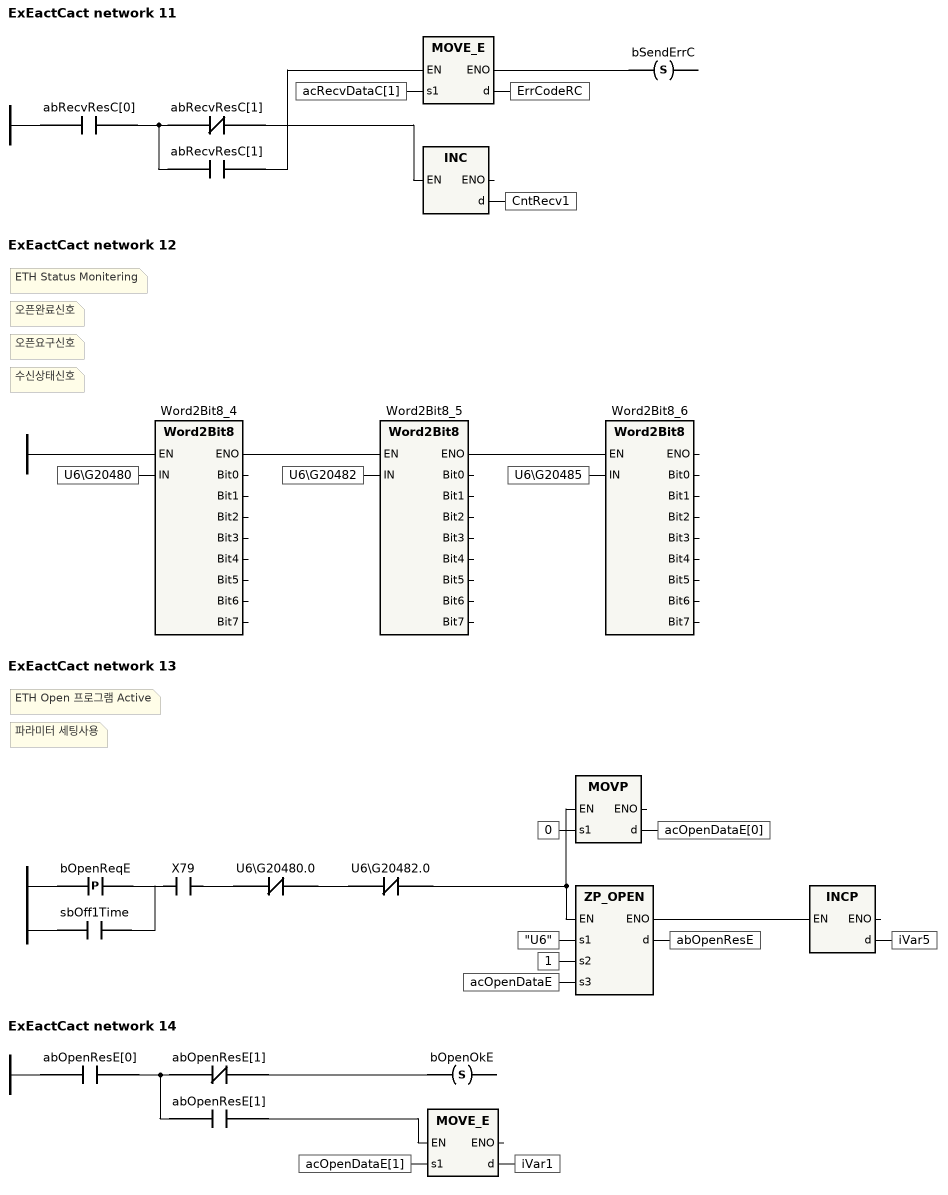
(* [picture p24: structured ladder/FBD of ExEactCact, networks 11 to 14] *)
(* network 11 *)
INC(abRecvResC[0] AND NOT abRecvResC[1], CntRecv1);
_e1 := MOVE_E(abRecvResC[0] AND abRecvResC[1], acRecvDataC[1], ErrCodeRC);
SET(_e1, bSendErrC);
(* network 12 *)
(* ETH Status Monitering *)
(* 오픈완료신호 *)
(* 오픈요구신호 *)
(* 수신상태신호 *)
Word2Bit8_4(EN := TRUE, IN := U6\G20480);
Word2Bit8_5(EN := Word2Bit8_4.ENO, IN := U6\G20482);
Word2Bit8_6(EN := Word2Bit8_5.ENO, IN := U6\G20485);
(* network 13 *)
(* ETH Open 프로그램 Active *)
(* 파라미터 세팅사용 *)
_p1 := (((LDP(TRUE, bOpenReqE) OR sbOff1Time) AND X79) AND NOT U6\G20480.0) AND NOT U6\G20482.0;
MOVP(_p1, 0, acOpenDataE[0]);
_e2 := ZP_OPEN(_p1, "U6", 1, acOpenDataE, abOpenResE);
INCP(_e2, iVar5);
(* network 14 *)
SET(abOpenResE[0] AND NOT abOpenResE[1], bOpenOkE);
MOVE_E(abOpenResE[0] AND abOpenResE[1], acOpenDataE[1], iVar1);
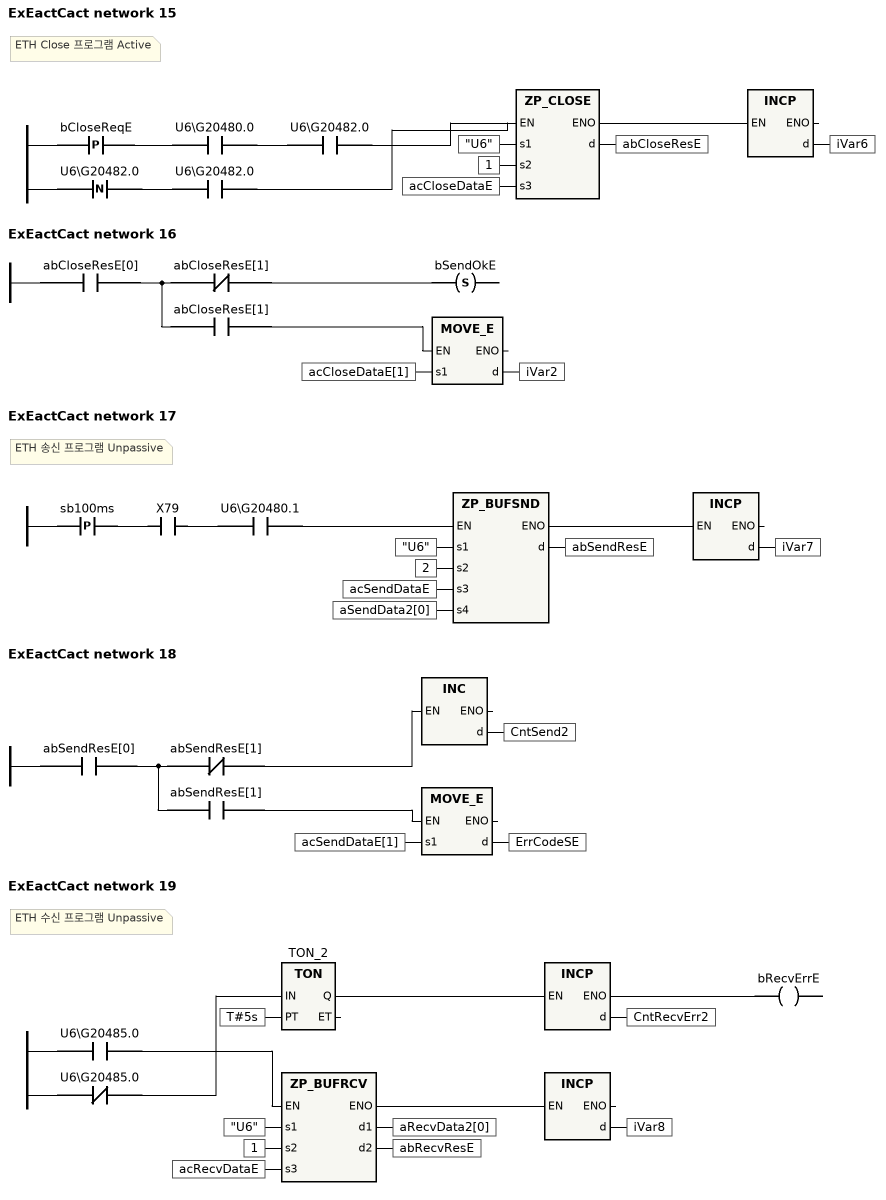
(* network 15 *)
(* ETH Close 프로그램 Active *)
_e1 := ZP_CLOSE((LDP(TRUE, bCloseReqE) AND U6\G20480.0 AND U6\G20482.0) OR (LDF(TRUE, U6\G20482.0) AND U6\G20482.0), "U6", 1, acCloseDataE, abCloseResE);
INCP(_e1, iVar6);
(* network 16 *)
SET(abCloseResE[0] AND NOT abCloseResE[1], bSendOkE);
MOVE_E(abCloseResE[0] AND abCloseResE[1], acCloseDataE[1], iVar2);
(* network 17 *)
(* ETH 송신 프로그램 Unpassive *)
_e1 := ZP_BUFSND(LDP(TRUE, sb100ms) AND X79 AND U6\G20480.1, "U6", 2, acSendDataE, aSendData2[0], abSendResE);
INCP(_e1, iVar7);
(* network 18 *)
INC(abSendResE[0] AND NOT abSendResE[1], CntSend2);
MOVE_E(abSendResE[0] AND abSendResE[1], acSendDataE[1], ErrCodeSE);
(* network 19 *)
(* ETH 수신 프로그램 Unpassive *)
_e1 := ZP_BUFRCV(U6\G20485.0, "U6", 1, acRecvDataE, aRecvData2[0], abRecvResE);
INCP(_e1, iVar8);
TON_2(IN := NOT U6\G20485.0, PT := T#5s);
_e2 := INCP(TON_2.Q, CntRecvErr2);
bRecvErrE := _e2;
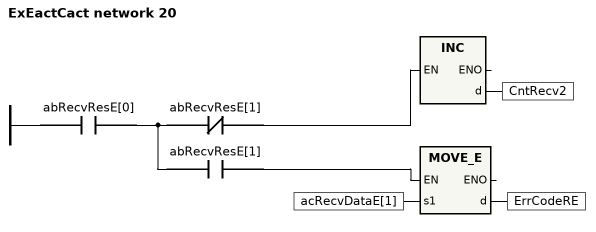
(* network 20 *)
INC(abRecvResE[0] AND NOT abRecvResE[1], CntRecv2);
MOVE_E(abRecvResE[0] AND abRecvResE[1], acRecvDataE[1], ErrCodeRE);
END_PROGRAM

PROGRAM ExEudpCudp
VAR
  bOpenReqC : BOOL;
  bCsetReq : BOOL;
  bOpenReqE : BOOL;
  bOpenOkC : BOOL;
  bOpenOkE : BOOL;
  bOpenErrC : BOOL;
  bOpenErrE : BOOL;
  abOpenResC : ARRAY [0..1] OF BOOL;
  abOpenResE : ARRAY [0..1] OF BOOL;
  acOpenDataC : ARRAY [0..9] OF INT;
  acCsetData : ARRAY [0..4] OF INT;
  acRdCtrl : ARRAY [0..9] OF INT;
  bSendReqC : BOOL;
  bSendReqE : BOOL;
  bSendOkC : BOOL;
  bSendOkE : BOOL;
  bSendErrC : BOOL;
  bSendErrE : BOOL;
  abSendResC : ARRAY [0..1] OF BOOL;
  abSendResE : ARRAY [0..1] OF BOOL;
  abSendResF : ARRAY [0..1] OF BOOL;
  acSendDataC : ARRAY [0..1] OF INT;
  acSendDataE : ARRAY [0..1] OF INT;
  acSendDataF : ARRAY [0..1] OF INT;
  bRecvOkC : BOOL;
  bRecvOkE : BOOL;
  bRecvOkF : BOOL;
  bRecvErrC : BOOL;
  bRecvErrE : BOOL;
  bRecvErrF : BOOL;
  abRecvResC : ARRAY [0..1] OF BOOL;
  abRecvRes3 : ARRAY [0..1] OF BOOL;
  abRecvRes13 : ARRAY [0..1] OF BOOL;
  acRecvDataC : ARRAY [0..1] OF INT;
  acRecvData3 : ARRAY [0..1] OF INT;
  acRecvData13 : ARRAY [0..1] OF INT;
  bCloseReqC : BOOL;
  bCloseOkC : BOOL;
  bCloseOkE : BOOL;
  bCloseErrC : BOOL;
  bCloseErrE : BOOL;
  abCloseResC : ARRAY [0..1] OF BOOL;
  abCloseResE : ARRAY [0..1] OF BOOL;
  acCloseDataC : ARRAY [0..1] OF INT;
  CntSend1 : INT;
  CntSend2 : INT;
  CntSend3 : INT;
  CntRecv1 : INT;
  CntRecvErr1 : INT;
  CntRecv2 : INT;
  CntRecv3 : INT;
  CntRecvErr2 : INT;
  CntRecvErr3 : INT;
  ErrCodeSC : INT;
  ErrCodeSE : INT;
  ErrCodeSF : INT;
  ErrCodeRC : INT;
  ErrCodeR3 : INT;
  ErrCodeR13 : INT;
  Mov4INT_1 : Mov4INT;
  Mov8INT_1 : Mov8INT;
  Mov4INT_2 : Mov4INT;
  Mov4INT_3 : Mov4INT;
  Mov4INT_4 : Mov4INT;
  Word2Bit8_1 : Word2Bit8;
  Word2Bit8_2 : Word2Bit8;
  Word2Bit8_3 : Word2Bit8;
  Word2Bit8_4 : Word2Bit8;
  Word2Bit8_5 : Word2Bit8;
  Word2Bit8_6 : Word2Bit8;
  TON_1 : TON;
  TON_2 : TON;
  TON_3 : TON;
  bCloseReqE : BOOL;
  acOpenDataE : ARRAY [0..9] OF INT;
  acCloseDataE : ARRAY [0..1] OF INT;
  ErrCodeOC : INT;
  ErrCodeOE : INT;
  ErrCodeCC : INT;
  ErrCodeCE : INT;
  bDelay : BOOL;
  bLedOff : BOOL;
  bChgReq : BOOL;
  bChgConn : BOOL;
  ChgPort : INT;
  CntRecv13 : INT;
  TON_13 : TON;
END_VAR
(* structured ladder/FBD written out as ST: instructions are called as NAME(EN, inputs, outputs); _pN, _eN, _tN stand for wires *)
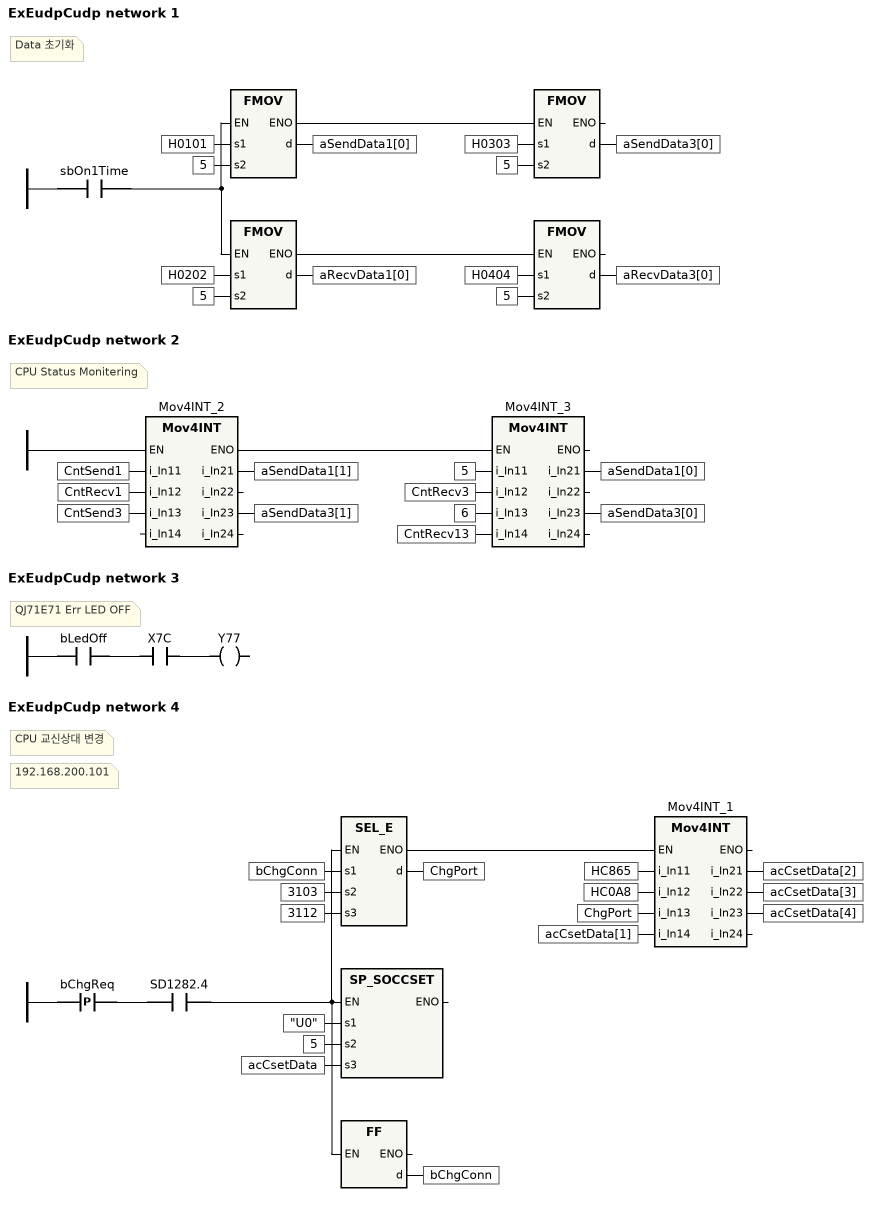
(* network 1 *)
(* Data 초기화 *)
_e1 := FMOV(sbOn1Time, H0101, 5, aSendData1[0]);
FMOV(_e1, H0303, 5, aSendData3[0]);
_e2 := FMOV(sbOn1Time, H0202, 5, aRecvData1[0]);
FMOV(_e2, H0404, 5, aRecvData3[0]);
(* network 2 *)
(* CPU Status Monitering *)
Mov4INT_2(EN := TRUE, i_In11 := CntSend1, i_In12 := CntRecv1, i_In13 := CntSend3, i_In21 => aSendData1[1], i_In23 => aSendData3[1]);
Mov4INT_3(EN := Mov4INT_2.ENO, i_In11 := 5, i_In12 := CntRecv3, i_In13 := 6, i_In14 := CntRecv13, i_In21 => aSendData1[0], i_In23 => aSendData3[0]);
(* network 3 *)
(* QJ71E71 Err LED OFF *)
Y77 := bLedOff AND X7C;
(* network 4 *)
(* CPU 교신상대 변경 *)
(* 192.168.200.101 *)
_p1 := LDP(TRUE, bChgReq) AND SD1282.4;
_e2 := SEL_E(_p1, bChgConn, 3103, 3112, ChgPort);
Mov4INT_1(EN := _e2, i_In11 := HC865, i_In12 := HC0A8, i_In13 := ChgPort, i_In14 := acCsetData[1], i_In21 => acCsetData[2], i_In22 => acCsetData[3], i_In23 => acCsetData[4]);
SP_SOCCSET(_p1, "U0", 5, acCsetData);
FF(_p1, bChgConn);
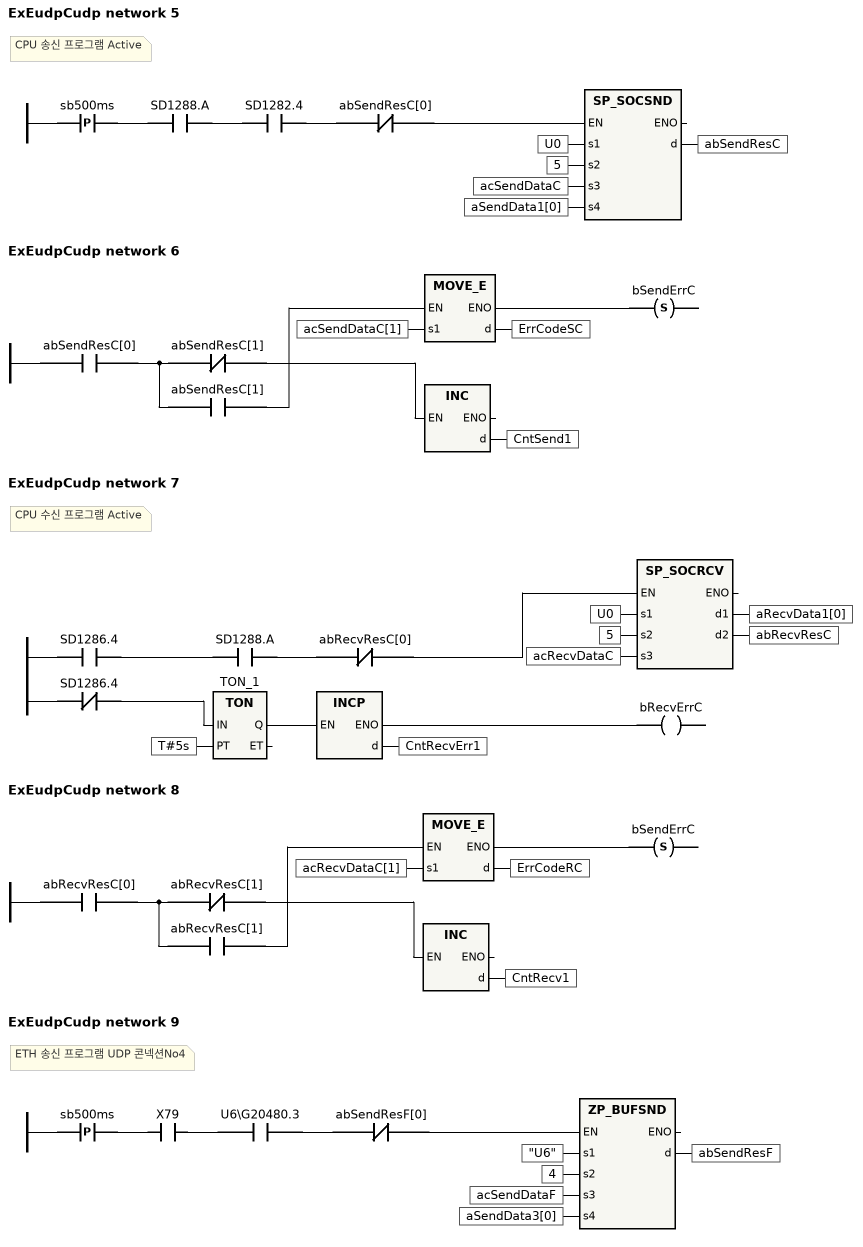
(* network 5 *)
(* CPU 송신 프로그램 Active *)
SP_SOCSND(LDP(TRUE, sb500ms) AND SD1288.A AND SD1282.4 AND NOT abSendResC[0], U0, 5, acSendDataC, aSendData1[0], abSendResC);
(* network 6 *)
INC(abSendResC[0] AND NOT abSendResC[1], CntSend1);
_e1 := MOVE_E(abSendResC[0] AND abSendResC[1], acSendDataC[1], ErrCodeSC);
SET(_e1, bSendErrC);
(* network 7 *)
(* CPU 수신 프로그램 Active *)
SP_SOCRCV(SD1286.4 AND SD1288.A AND NOT abRecvResC[0], U0, 5, acRecvDataC, aRecvData1[0], abRecvResC);
TON_1(IN := NOT SD1286.4, PT := T#5s);
_e1 := INCP(TON_1.Q, CntRecvErr1);
bRecvErrC := _e1;
(* network 8 *)
INC(abRecvResC[0] AND NOT abRecvResC[1], CntRecv1);
_e1 := MOVE_E(abRecvResC[0] AND abRecvResC[1], acRecvDataC[1], ErrCodeRC);
SET(_e1, bSendErrC);
(* network 9 *)
(* ETH 송신 프로그램 UDP 콘넥션No4 *)
ZP_BUFSND(LDP(TRUE, sb500ms) AND X79 AND U6\G20480.3 AND NOT abSendResF[0], "U6", 4, acSendDataF, aSendData3[0], abSendResF);
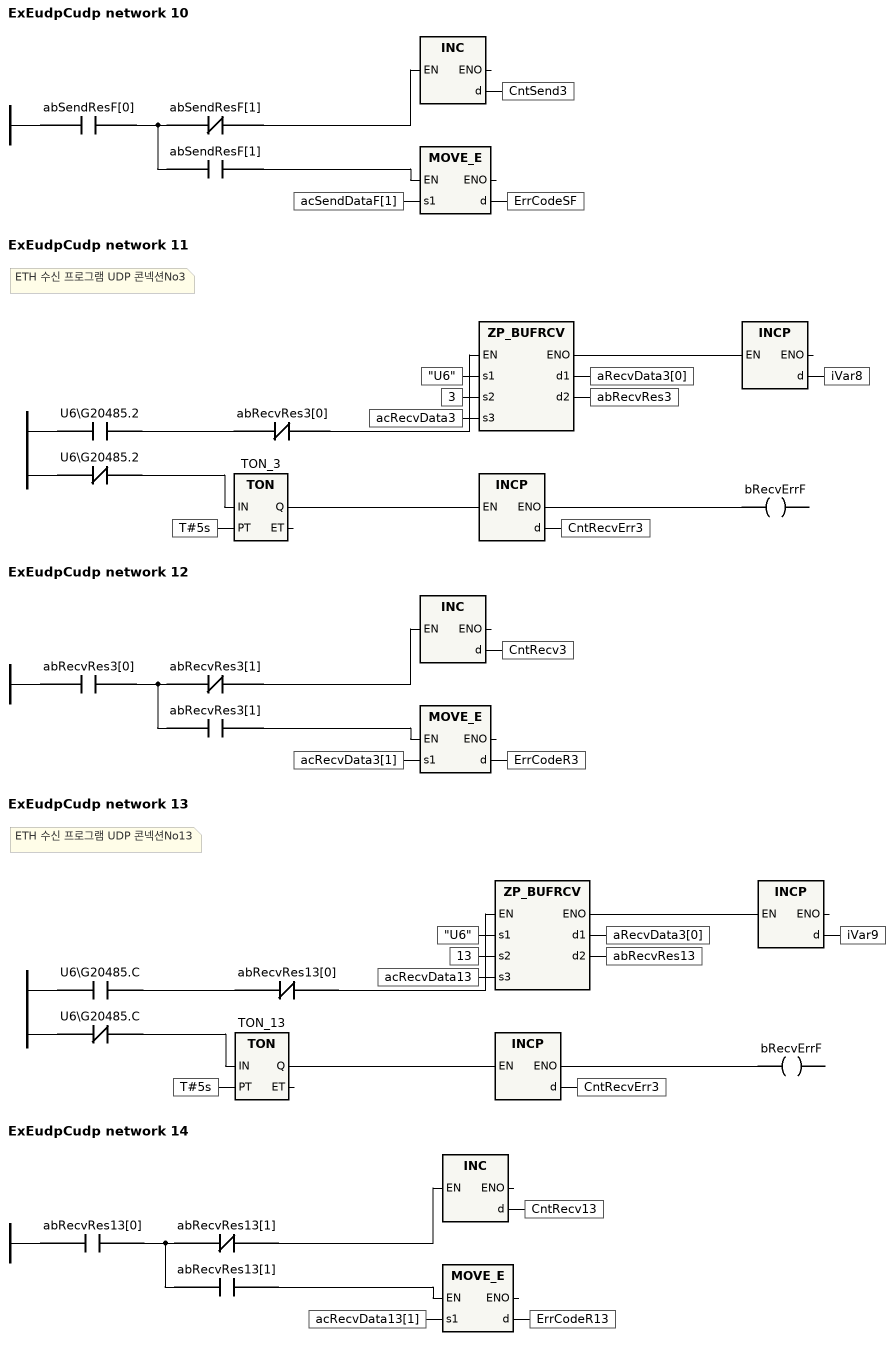
(* network 10 *)
INC(abSendResF[0] AND NOT abSendResF[1], CntSend3);
MOVE_E(abSendResF[0] AND abSendResF[1], acSendDataF[1], ErrCodeSF);
(* network 11 *)
(* ETH 수신 프로그램 UDP 콘넥션No3 *)
_e1 := ZP_BUFRCV(U6\G20485.2 AND NOT abRecvRes3[0], "U6", 3, acRecvData3, aRecvData3[0], abRecvRes3);
INCP(_e1, iVar8);
TON_3(IN := NOT U6\G20485.2, PT := T#5s);
_e2 := INCP(TON_3.Q, CntRecvErr3);
bRecvErrF := _e2;
(* network 12 *)
INC(abRecvRes3[0] AND NOT abRecvRes3[1], CntRecv3);
MOVE_E(abRecvRes3[0] AND abRecvRes3[1], acRecvData3[1], ErrCodeR3);
(* network 13 *)
(* ETH 수신 프로그램 UDP 콘넥션No13 *)
_e1 := ZP_BUFRCV(U6\G20485.C AND NOT abRecvRes13[0], "U6", 13, acRecvData13, aRecvData3[0], abRecvRes13);
INCP(_e1, iVar9);
TON_13(IN := NOT U6\G20485.C, PT := T#5s);
_e2 := INCP(TON_13.Q, CntRecvErr3);
bRecvErrF := _e2;
(* network 14 *)
INC(abRecvRes13[0] AND NOT abRecvRes13[1], CntRecv13);
MOVE_E(abRecvRes13[0] AND abRecvRes13[1], acRecvData13[1], ErrCodeR13);
END_PROGRAM

FUNCTION_BLOCK Word2Bit16
VAR_INPUT
  bEN : BOOL;
END_VAR
VAR_OUTPUT
  Bit0 : BOOL;
  Bit1 : BOOL;
  Bit2 : BOOL;
  Bit3 : BOOL;
  Bit4 : BOOL;
  Bit5 : BOOL;
  Bit6 : BOOL;
  Bit7 : BOOL;
  Bit8 : BOOL;
  Bit9 : BOOL;
  Bit10 : BOOL;
  Bit11 : BOOL;
  Bit12 : BOOL;
  Bit13 : BOOL;
  Bit14 : BOOL;
  Bit15 : BOOL;
END_VAR
VAR_INPUT
  InWord : WORD;
END_VAR
VAR_OUTPUT
  bENO : BOOL;
END_VAR
VAR
  InVal : WORD;
END_VAR
 
bENO := bEN;
InVal :=InWord;
Bit0 := (InVal AND 16#0001) = H0001;
Bit1 := (InVal AND 16#0002) = H0002;
Bit2 := (InVal AND 16#0004) = H0004;
Bit3 := (InVal AND 16#0008) = H0008;
Bit4 := (InVal AND 16#0010) = H0010;
Bit5 := (InVal AND 16#0020) = H0020;
Bit6 := (InVal AND 16#0040) = H0040;
Bit7 := (InVal AND 16#0080) = H0080;
Bit8 := (InVal AND 16#0100) = H0100;
Bit9 := (InVal AND 16#0200) = H0200;
Bit10 := (InVal AND 16#0400) = H0400;
Bit11 := (InVal AND 16#0800) = H0800;
Bit12 := (InVal AND 16#1000) = H1000;
Bit13 := (InVal AND 16#2000) = H2000;
Bit14 := (InVal AND 16#4000) = H4000;
Bit15 := (InVal AND 16#8000) = H8000;

(*
Bit0 := WORD_TO_BOOL(IN AND 16#0001);
Bit1 := WORD_TO_BOOL(SHR(IN AND 16#0002 , 1));
Bit2 := WORD_TO_BOOL(SHR(IN AND 16#0004 , 2));
Bit3 := WORD_TO_BOOL(SHR(IN AND 16#0008 , 3));
Bit4 := WORD_TO_BOOL(SHR(IN AND 16#0010 , 4));
Bit5 := WORD_TO_BOOL(SHR(IN AND 16#0020 , 5));
Bit6 := WORD_TO_BOOL(SHR(IN AND 16#0040 , 6));
Bit7 := WORD_TO_BOOL(SHR(IN AND 16#0080 , 7));
 
Bit8 := WORD_TO_BOOL(SHR(IN AND 16#0100 , 8));
Bit9 := WORD_TO_BOOL(SHR(IN AND 16#0200 , 9));
Bit10 := WORD_TO_BOOL(SHR(IN AND 16#0400 , 10));
Bit11 := WORD_TO_BOOL(SHR(IN AND 16#0800 , 11));
Bit12 := WORD_TO_BOOL(SHR(IN AND 16#1000 , 12));
Bit13 := WORD_TO_BOOL(SHR(IN AND 16#2000 , 13));
Bit14 := WORD_TO_BOOL(SHR(IN AND 16#4000 , 14));
Bit15 := WORD_TO_BOOL(SHR(IN AND 16#8000 , 15));
*)
END_FUNCTION_BLOCK

PROGRAM ExEactCpas
VAR
  bOpenReqC : BOOL;
  bCsetReq : BOOL;
  bOpenReqE : BOOL;
  bOpenOkC : BOOL;
  bOpenOkE : BOOL;
  bOpenErrC : BOOL;
  bOpenErrE : BOOL;
  abOpenResC : ARRAY [0..1] OF BOOL;
  abOpenResE : ARRAY [0..1] OF BOOL;
  acOpenDataC : ARRAY [0..9] OF INT;
  acCsetData : ARRAY [0..4] OF INT;
  acRdCtrl : ARRAY [0..9] OF INT;
  bSendReqC : BOOL;
  bSendReqE : BOOL;
  bSendOkC : BOOL;
  bSendOkE : BOOL;
  bSendErrC : BOOL;
  bSendErrE : BOOL;
  abSendResC : ARRAY [0..1] OF BOOL;
  abSendResE : ARRAY [0..1] OF BOOL;
  abSendResF : ARRAY [0..1] OF BOOL;
  acSendDataC : ARRAY [0..1] OF INT;
  acSendDataE : ARRAY [0..1] OF INT;
  acSendDataF : ARRAY [0..1] OF INT;
  bRecvOkC : BOOL;
  bRecvOkE : BOOL;
  bRecvOkF : BOOL;
  bRecvErrC : BOOL;
  bRecvErrE : BOOL;
  bRecvErrF : BOOL;
  abRecvResC : ARRAY [0..1] OF BOOL;
  abRecvResE : ARRAY [0..1] OF BOOL;
  abRecvResF : ARRAY [0..1] OF BOOL;
  acRecvDataC : ARRAY [0..1] OF INT;
  acRecvDataE : ARRAY [0..1] OF INT;
  acRecvDataF : ARRAY [0..1] OF INT;
  bCloseReqC : BOOL;
  bCloseOkC : BOOL;
  bCloseOkE : BOOL;
  bCloseErrC : BOOL;
  bCloseErrE : BOOL;
  abCloseResC : ARRAY [0..1] OF BOOL;
  abCloseResE : ARRAY [0..1] OF BOOL;
  acCloseDataC : ARRAY [0..1] OF INT;
  CntSend1 : INT;
  CntSend2 : INT;
  CntSend3 : INT;
  CntRecv1 : INT;
  CntRecvErr1 : INT;
  CntRecv2 : INT;
  CntRecv3 : INT;
  CntRecvErr2 : INT;
  CntRecvErr3 : INT;
  ErrCodeCC : INT;
  ErrCodeSE : INT;
  ErrCodeSF : INT;
  ErrCodeRC : INT;
  ErrCodeRE : INT;
  ErrCodeRF : INT;
  Mov4INT_1 : Mov4INT;
  Mov8INT_1 : Mov8INT;
  Mov4INT_2 : Mov4INT;
  Mov4INT_3 : Mov4INT;
  Mov4INT_4 : Mov4INT;
  Word2Bit8_1 : Word2Bit8;
  Word2Bit8_2 : Word2Bit8;
  Word2Bit8_3 : Word2Bit8;
  Word2Bit8_4 : Word2Bit8;
  Word2Bit8_5 : Word2Bit8;
  Word2Bit8_6 : Word2Bit8;
  TON_1 : TON;
  TON_2 : TON;
  TON_3 : TON;
  Status1 : WORD;
  Status2 : WORD;
  Status3 : WORD;
  Word2Bit16_1 : Word2Bit16;
  Word2Bit16_2 : Word2Bit16;
  Word2Bit16_3 : Word2Bit16;
  acOpenDataE : ARRAY [0..9] OF INT;
  acCloseDataE : ARRAY [0..1] OF INT;
  ErrCodeOE : INT;
  ErrCodeSC : INT;
  ErrCodeCE : INT;
  ErrCodeOC : INT;
  bCloseReqE : BOOL;
  Mov4INT_5 : Mov4INT;
  Mov4INT_6 : Mov4INT;
  Mov4INT_7 : Mov4INT;
  Mov4INT_8 : Mov4INT;
END_VAR
(* structured ladder/FBD written out as ST: instructions are called as NAME(EN, inputs, outputs); _pN, _eN, _tN stand for wires *)
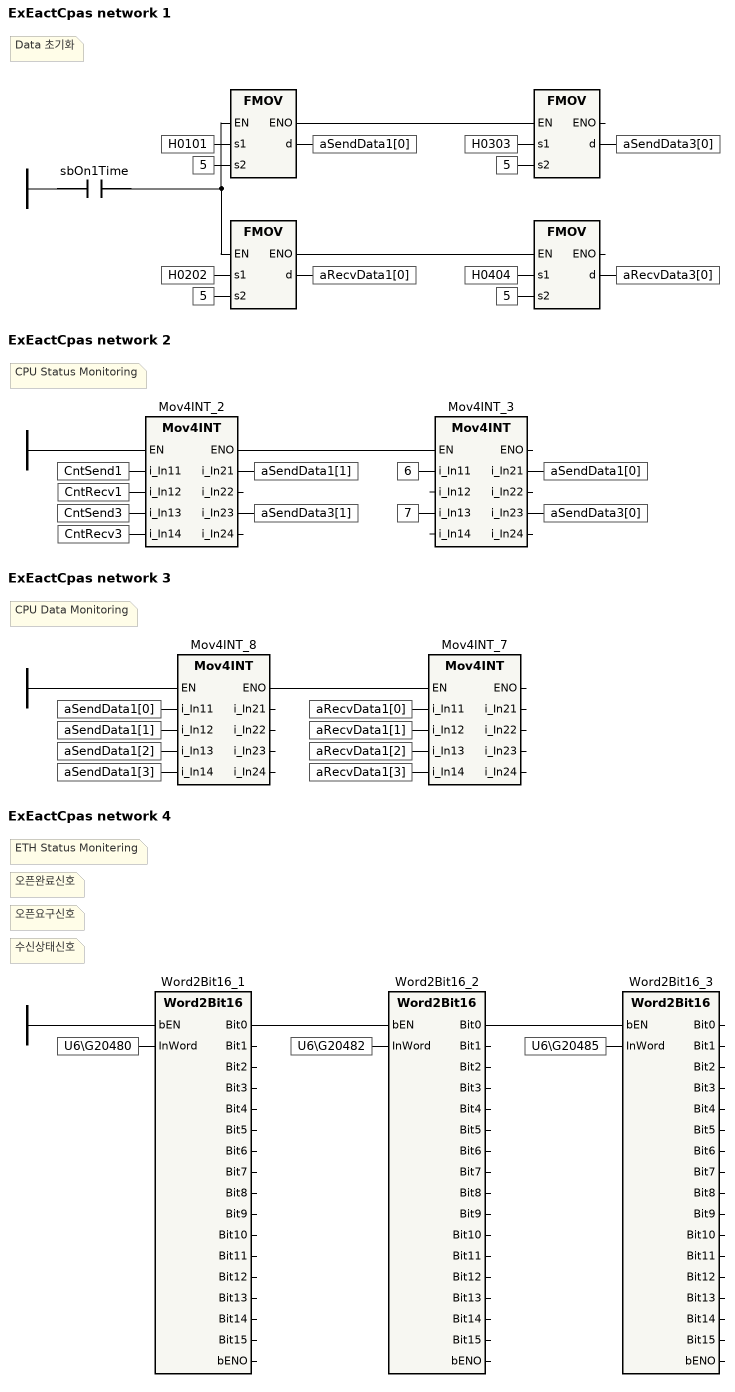
(* network 1 *)
(* Data 초기화 *)
_e1 := FMOV(sbOn1Time, H0101, 5, aSendData1[0]);
FMOV(_e1, H0303, 5, aSendData3[0]);
_e2 := FMOV(sbOn1Time, H0202, 5, aRecvData1[0]);
FMOV(_e2, H0404, 5, aRecvData3[0]);
(* network 2 *)
(* CPU Status Monitoring *)
Mov4INT_2(EN := TRUE, i_In11 := CntSend1, i_In12 := CntRecv1, i_In13 := CntSend3, i_In14 := CntRecv3, i_In21 => aSendData1[1], i_In23 => aSendData3[1]);
Mov4INT_3(EN := Mov4INT_2.ENO, i_In11 := 6, i_In13 := 7, i_In21 => aSendData1[0], i_In23 => aSendData3[0]);
(* network 3 *)
(* CPU Data Monitoring *)
Mov4INT_8(EN := TRUE, i_In11 := aSendData1[0], i_In12 := aSendData1[1], i_In13 := aSendData1[2], i_In14 := aSendData1[3]);
Mov4INT_7(EN := Mov4INT_8.ENO, i_In11 := aRecvData1[0], i_In12 := aRecvData1[1], i_In13 := aRecvData1[2], i_In14 := aRecvData1[3]);
(* network 4 *)
(* ETH Status Monitering *)
(* 오픈완료신호 *)
(* 오픈요구신호 *)
(* 수신상태신호 *)
Word2Bit16_1(bEN := TRUE, InWord := U6\G20480);
Word2Bit16_2(bEN := Word2Bit16_1.Bit0, InWord := U6\G20482);
Word2Bit16_3(bEN := Word2Bit16_2.Bit0, InWord := U6\G20485);
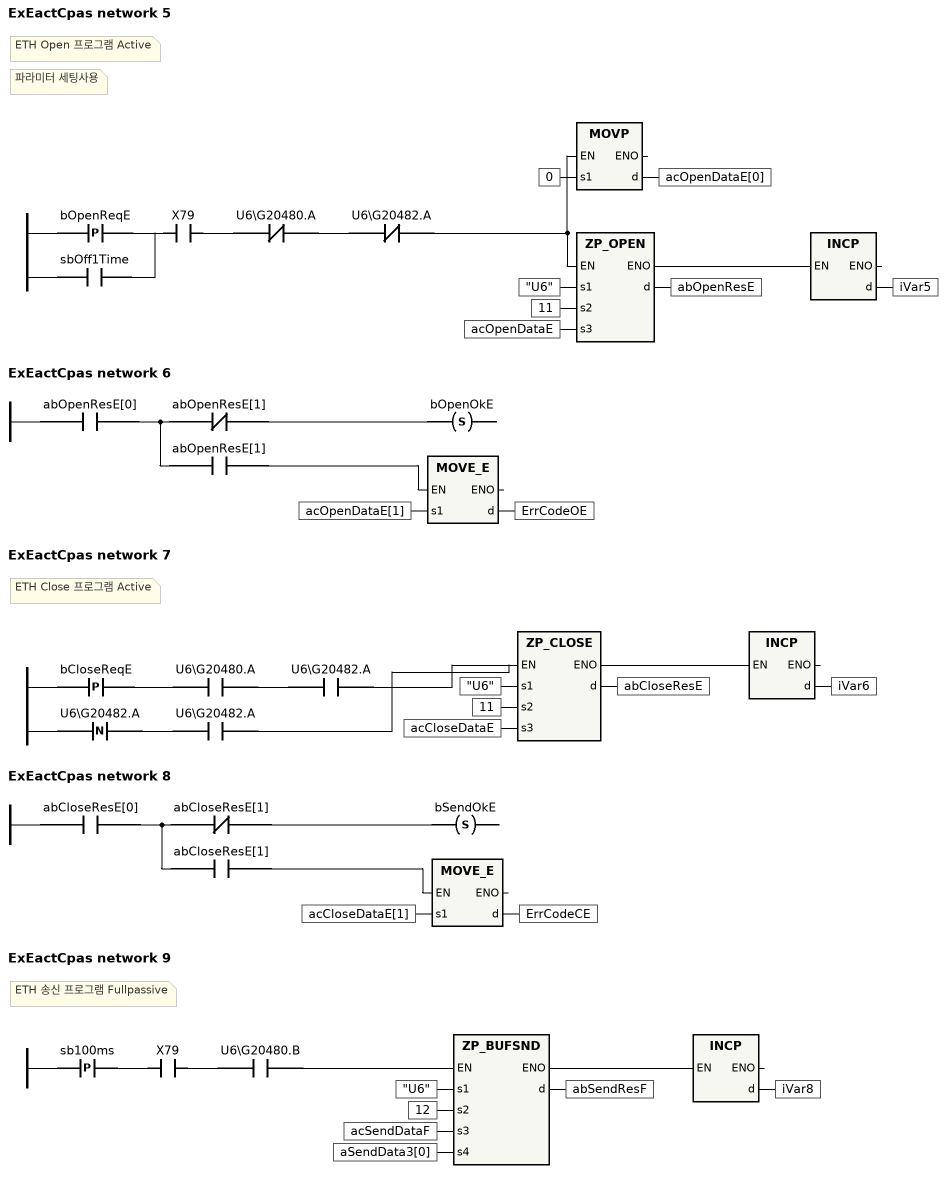
(* network 5 *)
(* ETH Open 프로그램 Active *)
(* 파라미터 세팅사용 *)
_p1 := (((LDP(TRUE, bOpenReqE) OR sbOff1Time) AND X79) AND NOT U6\G20480.A) AND NOT U6\G20482.A;
MOVP(_p1, 0, acOpenDataE[0]);
_e2 := ZP_OPEN(_p1, "U6", 11, acOpenDataE, abOpenResE);
INCP(_e2, iVar5);
(* network 6 *)
SET(abOpenResE[0] AND NOT abOpenResE[1], bOpenOkE);
MOVE_E(abOpenResE[0] AND abOpenResE[1], acOpenDataE[1], ErrCodeOE);
(* network 7 *)
(* ETH Close 프로그램 Active *)
_e1 := ZP_CLOSE((LDP(TRUE, bCloseReqE) AND U6\G20480.A AND U6\G20482.A) OR (LDF(TRUE, U6\G20482.A) AND U6\G20482.A), "U6", 11, acCloseDataE, abCloseResE);
INCP(_e1, iVar6);
(* network 8 *)
SET(abCloseResE[0] AND NOT abCloseResE[1], bSendOkE);
MOVE_E(abCloseResE[0] AND abCloseResE[1], acCloseDataE[1], ErrCodeCE);
(* network 9 *)
(* ETH 송신 프로그램 Fullpassive *)
_e1 := ZP_BUFSND(LDP(TRUE, sb100ms) AND X79 AND U6\G20480.B, "U6", 12, acSendDataF, aSendData3[0], abSendResF);
INCP(_e1, iVar8);
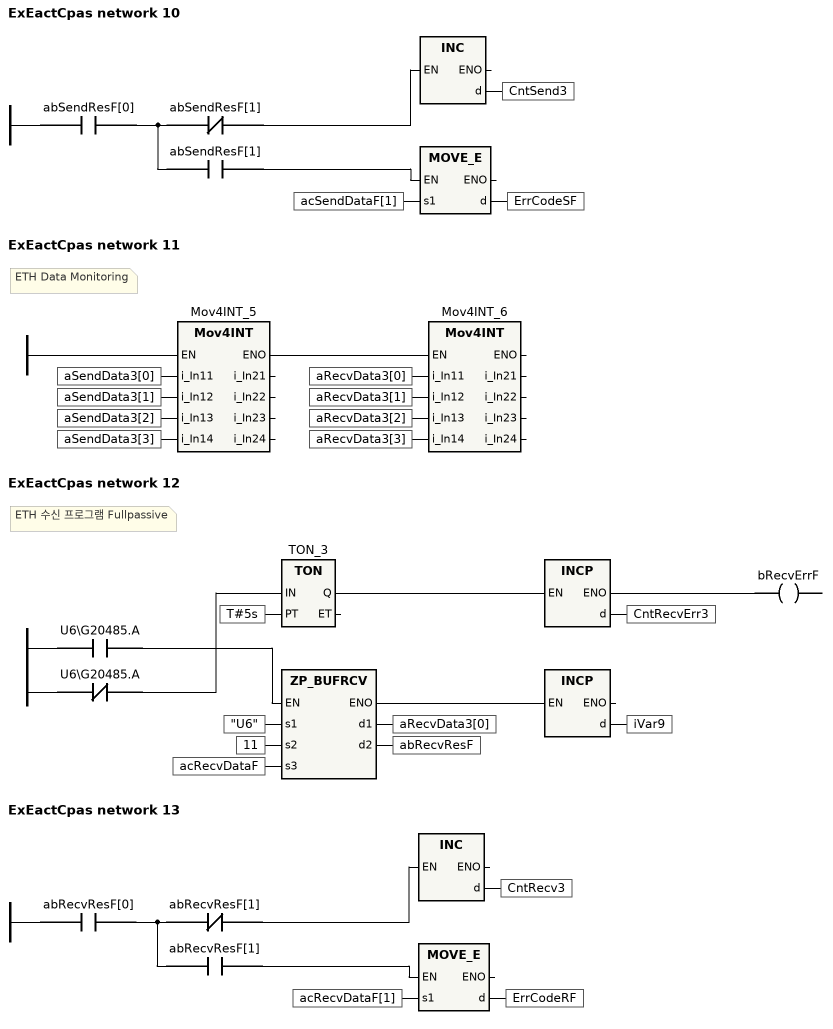
(* network 10 *)
INC(abSendResF[0] AND NOT abSendResF[1], CntSend3);
MOVE_E(abSendResF[0] AND abSendResF[1], acSendDataF[1], ErrCodeSF);
(* network 11 *)
(* ETH Data Monitoring *)
Mov4INT_5(EN := TRUE, i_In11 := aSendData3[0], i_In12 := aSendData3[1], i_In13 := aSendData3[2], i_In14 := aSendData3[3]);
Mov4INT_6(EN := Mov4INT_5.ENO, i_In11 := aRecvData3[0], i_In12 := aRecvData3[1], i_In13 := aRecvData3[2], i_In14 := aRecvData3[3]);
(* network 12 *)
(* ETH 수신 프로그램 Fullpassive *)
_e1 := ZP_BUFRCV(U6\G20485.A, "U6", 11, acRecvDataF, aRecvData3[0], abRecvResF);
INCP(_e1, iVar9);
TON_3(IN := NOT U6\G20485.A, PT := T#5s);
_e2 := INCP(TON_3.Q, CntRecvErr3);
bRecvErrF := _e2;
(* network 13 *)
INC(abRecvResF[0] AND NOT abRecvResF[1], CntRecv3);
MOVE_E(abRecvResF[0] AND abRecvResF[1], acRecvDataF[1], ErrCodeRF);
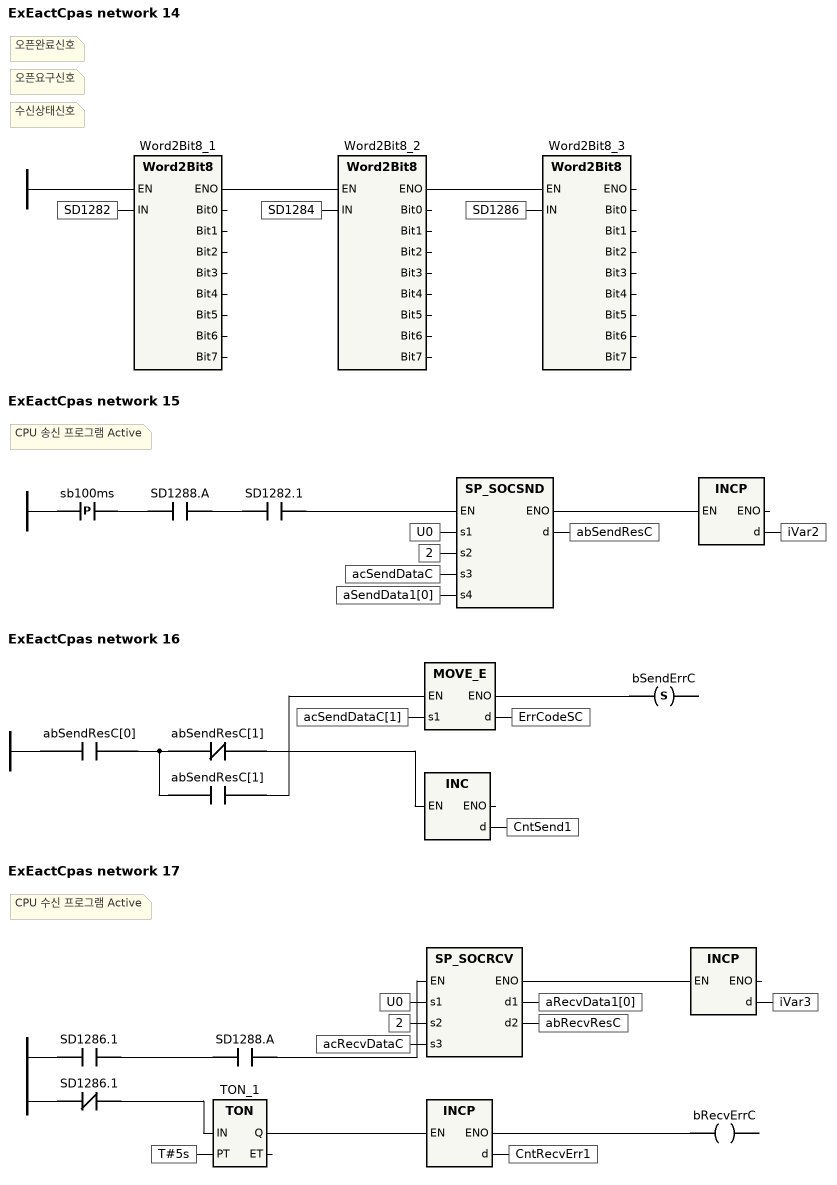
(* network 14 *)
(* 오픈완료신호 *)
(* 오픈요구신호 *)
(* 수신상태신호 *)
Word2Bit8_1(EN := TRUE, IN := SD1282);
Word2Bit8_2(EN := Word2Bit8_1.ENO, IN := SD1284);
Word2Bit8_3(EN := Word2Bit8_2.ENO, IN := SD1286);
(* network 15 *)
(* CPU 송신 프로그램 Active *)
_e1 := SP_SOCSND(LDP(TRUE, sb100ms) AND SD1288.A AND SD1282.1, U0, 2, acSendDataC, aSendData1[0], abSendResC);
INCP(_e1, iVar2);
(* network 16 *)
INC(abSendResC[0] AND NOT abSendResC[1], CntSend1);
_e1 := MOVE_E(abSendResC[0] AND abSendResC[1], acSendDataC[1], ErrCodeSC);
SET(_e1, bSendErrC);
(* network 17 *)
(* CPU 수신 프로그램 Active *)
_e1 := SP_SOCRCV(SD1286.1 AND SD1288.A, U0, 2, acRecvDataC, aRecvData1[0], abRecvResC);
INCP(_e1, iVar3);
TON_1(IN := NOT SD1286.1, PT := T#5s);
_e2 := INCP(TON_1.Q, CntRecvErr1);
bRecvErrC := _e2;
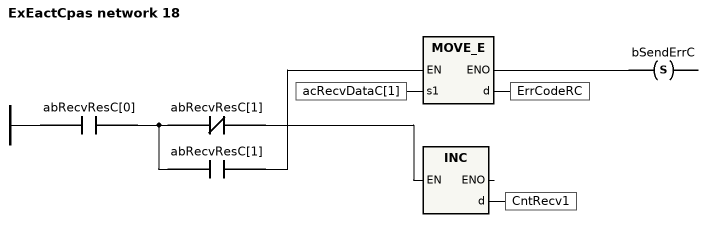
(* network 18 *)
INC(abRecvResC[0] AND NOT abRecvResC[1], CntRecv1);
_e1 := MOVE_E(abRecvResC[0] AND abRecvResC[1], acRecvDataC[1], ErrCodeRC);
SET(_e1, bSendErrC);
END_PROGRAM

PROGRAM ExZP_OPEN
VAR
  bOpenExeE : BOOL;
  bOpenOkE : BOOL;
  bOpenErrE : BOOL;
  bComp11 : BOOL;
  bReq11 : BOOL;
  acOpenDataE : ARRAY [0..9] OF INT;
  bCloseTime : BOOL;
  bCloseReqE : BOOL;
  bCloseExeE : BOOL;
  bCloseReqA : BOOL;
  bCloseIng : BOOL;
  acCloseDataE : ARRAY [0..1] OF INT;
  abOpenResE : ARRAY [0..1] OF BOOL;
  abCloseResE : ARRAY [0..1] OF BOOL;
  bCloseOkE : BOOL;
  bCloseErrE : BOOL;
  bOpenReqM : BOOL;
  bCloseReqM : BOOL;
  Word2Bit16_1 : Word2Bit16;
  Word2Bit16_2 : Word2Bit16;
  Word2Bit16_3 : Word2Bit16;
  abSendResE : ARRAY [0..1] OF BOOL;
  acSendDataE : ARRAY [0..1] OF INT;
  Mov4INT_1 : Mov4INT;
  bReqFlag : BOOL;
  bFlagExe : BOOL;
  bReqOpen : BOOL;
END_VAR
(* structured ladder/FBD written out as ST: instructions are called as NAME(EN, inputs, outputs); _pN, _eN, _tN stand for wires *)
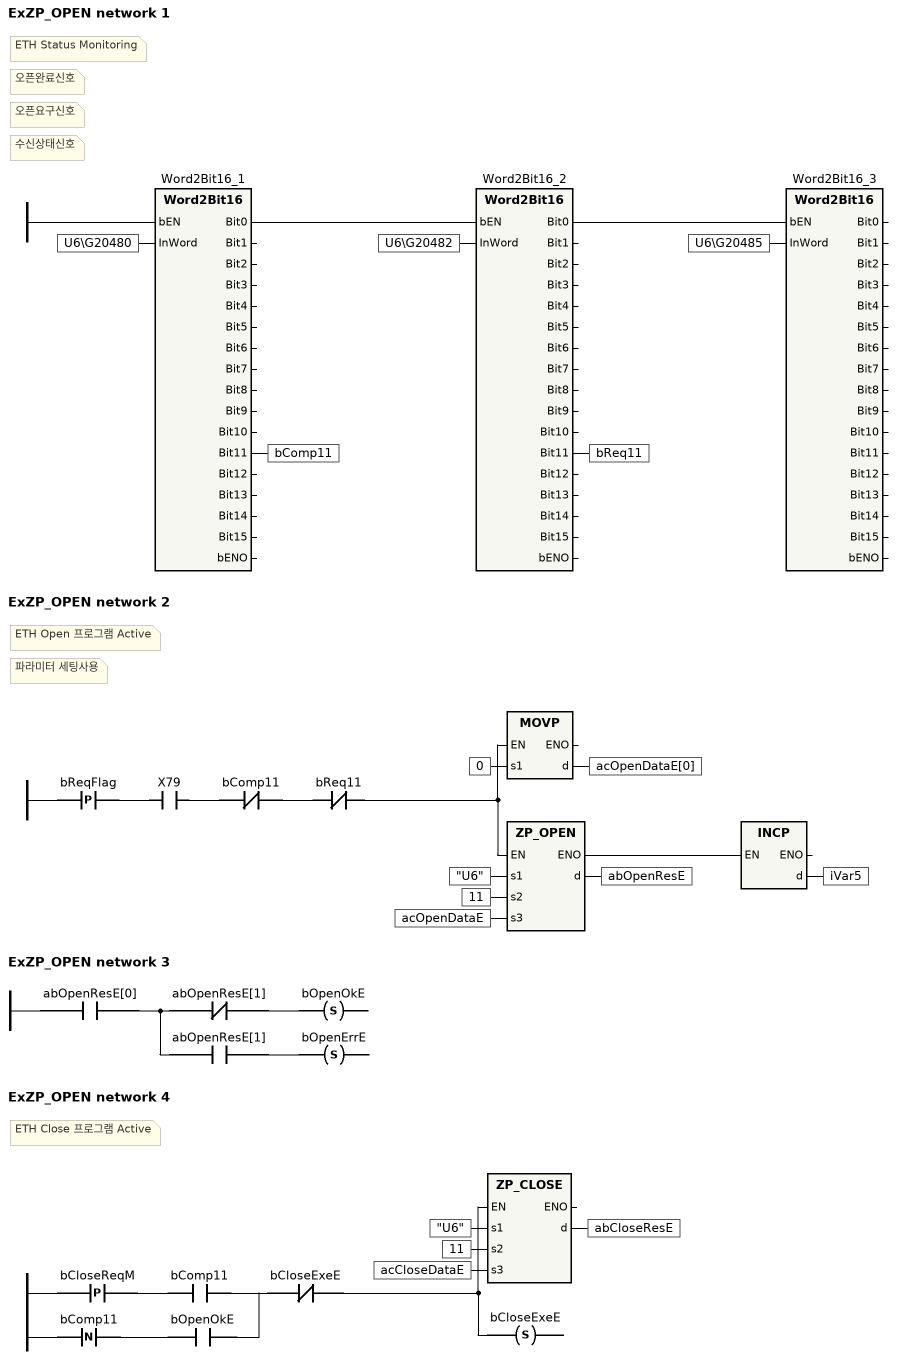
(* network 1 *)
(* ETH Status Monitoring *)
(* 오픈완료신호 *)
(* 오픈요구신호 *)
(* 수신상태신호 *)
Word2Bit16_1(bEN := TRUE, InWord := U6\G20480, Bit11 => bComp11);
Word2Bit16_2(bEN := Word2Bit16_1.Bit0, InWord := U6\G20482, Bit11 => bReq11);
Word2Bit16_3(bEN := Word2Bit16_2.Bit0, InWord := U6\G20485);
(* network 2 *)
(* ETH Open 프로그램 Active *)
(* 파라미터 세팅사용 *)
_p1 := LDP(TRUE, bReqFlag) AND X79 AND NOT bComp11 AND NOT bReq11;
MOVP(_p1, 0, acOpenDataE[0]);
_e2 := ZP_OPEN(_p1, "U6", 11, acOpenDataE, abOpenResE);
INCP(_e2, iVar5);
(* network 3 *)
SET(abOpenResE[0] AND NOT abOpenResE[1], bOpenOkE);
SET(abOpenResE[0] AND abOpenResE[1], bOpenErrE);
(* network 4 *)
(* ETH Close 프로그램 Active *)
_p1 := ((LDP(TRUE, bCloseReqM) AND bComp11) OR (LDF(TRUE, bComp11) AND bOpenOkE)) AND NOT bCloseExeE;
ZP_CLOSE(_p1, "U6", 11, acCloseDataE, abCloseResE);
SET(_p1, bCloseExeE);
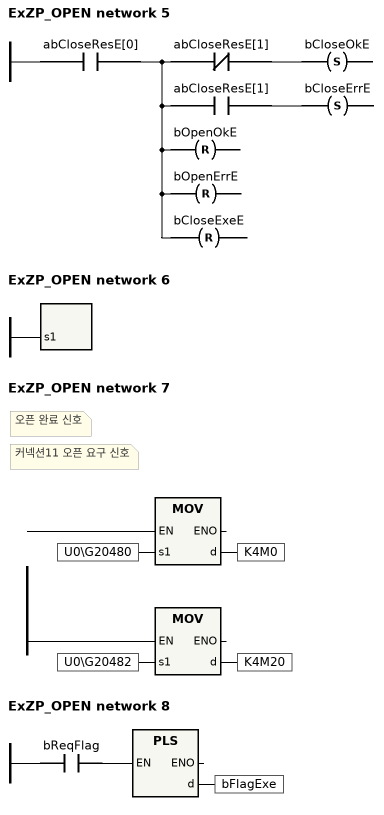
(* network 5 *)
SET(abCloseResE[0] AND NOT abCloseResE[1], bCloseOkE);
SET(abCloseResE[0] AND abCloseResE[1], bCloseErrE);
RST(abCloseResE[0], bOpenOkE);
RST(abCloseResE[0], bOpenErrE);
RST(abCloseResE[0], bCloseExeE);
(* network 6 *)
(* element kind 10  <- TRUE *)
(* network 7 *)
(* 오픈 완료 신호 *)
(* 커넥션11 오픈 요구 신호 *)
MOV(TRUE, U0\G20480, K4M0);
MOV(TRUE, U0\G20482, K4M20);
(* network 8 *)
PLS(bReqFlag, bFlagExe);
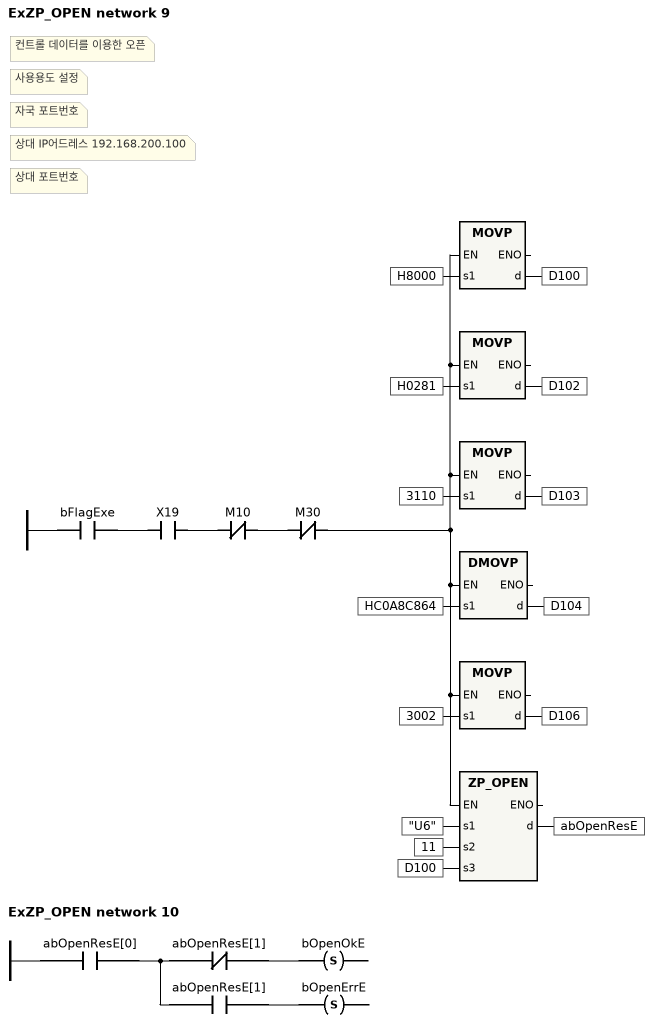
(* network 9 *)
(* 컨트롤 데이터를 이용한 오픈 *)
(* 사용용도 설정 *)
(* 자국 포트번호 *)
(* 상대 IP어드레스 192.168.200.100 *)
(* 상대 포트번호 *)
_p1 := bFlagExe AND X19 AND NOT M10 AND NOT M30;
MOVP(_p1, H8000, D100);
MOVP(_p1, H0281, D102);
MOVP(_p1, 3110, D103);
DMOVP(_p1, HC0A8C864, D104);
MOVP(_p1, 3002, D106);
ZP_OPEN(_p1, "U6", 11, D100, abOpenResE);
(* network 10 *)
SET(abOpenResE[0] AND NOT abOpenResE[1], bOpenOkE);
SET(abOpenResE[0] AND abOpenResE[1], bOpenErrE);
END_PROGRAM

PROGRAM xEx_ZP_CLOSE
VAR
  bOpenExeE : BOOL;
  bOpenOkE : BOOL;
  bOpenErrE : BOOL;
  bComp11 : BOOL;
  bReq11 : BOOL;
  acOpenDataE : ARRAY [0..9] OF INT;
  bCloseTime : BOOL;
  bCloseReqE : BOOL;
  bCloseExeE : BOOL;
  bCloseReqA : BOOL;
  bCloseIng : BOOL;
  acCloseDataE : ARRAY [0..1] OF INT;
  abOpenResE : ARRAY [0..1] OF BOOL;
  abCloseResE : ARRAY [0..1] OF BOOL;
  bCloseOkE : BOOL;
  bCloseErrE : BOOL;
  bOpenReqM : BOOL;
  bCloseReqM : BOOL;
  Word2Bit16_1 : Word2Bit16;
  Word2Bit16_2 : Word2Bit16;
  Word2Bit16_3 : Word2Bit16;
  abSendResE : ARRAY [0..1] OF BOOL;
  acSendDataE : ARRAY [0..1] OF INT;
  Mov4INT_1 : Mov4INT;
  bReqFlag : BOOL;
  bFlagExe : BOOL;
  bReqOpen : BOOL;
END_VAR
(* structured ladder/FBD written out as ST: instructions are called as NAME(EN, inputs, outputs); _pN, _eN, _tN stand for wires *)
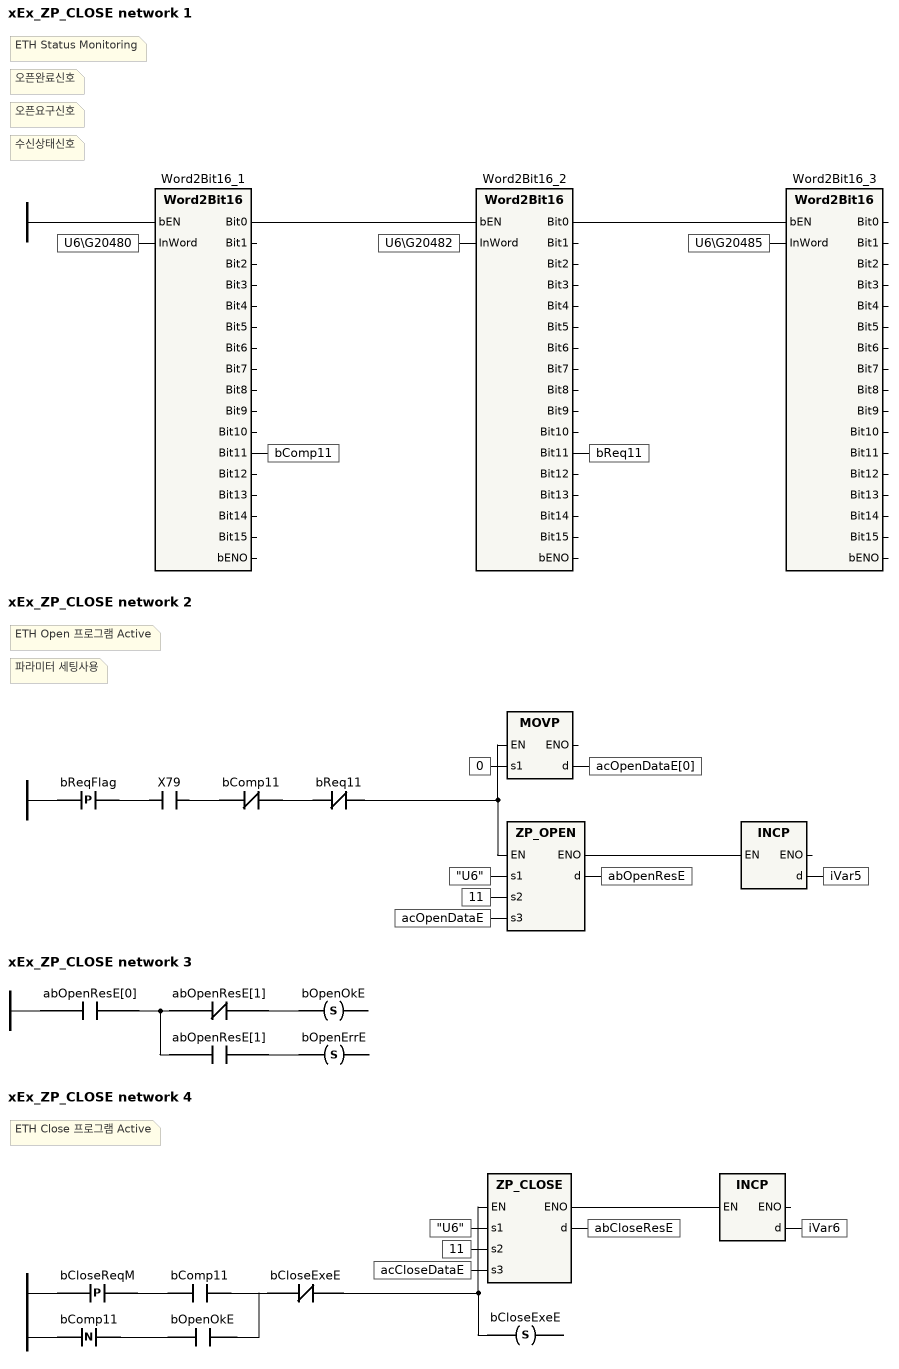
(* network 1 *)
(* ETH Status Monitoring *)
(* 오픈완료신호 *)
(* 오픈요구신호 *)
(* 수신상태신호 *)
Word2Bit16_1(bEN := TRUE, InWord := U6\G20480, Bit11 => bComp11);
Word2Bit16_2(bEN := Word2Bit16_1.Bit0, InWord := U6\G20482, Bit11 => bReq11);
Word2Bit16_3(bEN := Word2Bit16_2.Bit0, InWord := U6\G20485);
(* network 2 *)
(* ETH Open 프로그램 Active *)
(* 파라미터 세팅사용 *)
_p1 := LDP(TRUE, bReqFlag) AND X79 AND NOT bComp11 AND NOT bReq11;
MOVP(_p1, 0, acOpenDataE[0]);
_e2 := ZP_OPEN(_p1, "U6", 11, acOpenDataE, abOpenResE);
INCP(_e2, iVar5);
(* network 3 *)
SET(abOpenResE[0] AND NOT abOpenResE[1], bOpenOkE);
SET(abOpenResE[0] AND abOpenResE[1], bOpenErrE);
(* network 4 *)
(* ETH Close 프로그램 Active *)
_p1 := ((LDP(TRUE, bCloseReqM) AND bComp11) OR (LDF(TRUE, bComp11) AND bOpenOkE)) AND NOT bCloseExeE;
_e2 := ZP_CLOSE(_p1, "U6", 11, acCloseDataE, abCloseResE);
INCP(_e2, iVar6);
SET(_p1, bCloseExeE);
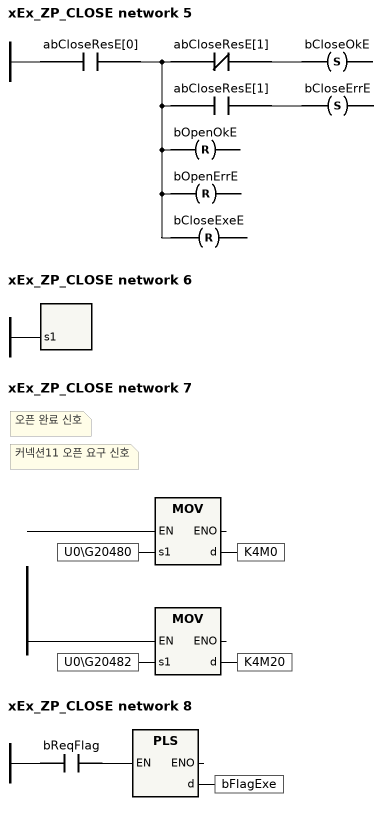
(* network 5 *)
SET(abCloseResE[0] AND NOT abCloseResE[1], bCloseOkE);
SET(abCloseResE[0] AND abCloseResE[1], bCloseErrE);
RST(abCloseResE[0], bOpenOkE);
RST(abCloseResE[0], bOpenErrE);
RST(abCloseResE[0], bCloseExeE);
(* network 6 *)
(* element kind 10  <- TRUE *)
(* network 7 *)
(* 오픈 완료 신호 *)
(* 커넥션11 오픈 요구 신호 *)
MOV(TRUE, U0\G20480, K4M0);
MOV(TRUE, U0\G20482, K4M20);
(* network 8 *)
PLS(bReqFlag, bFlagExe);
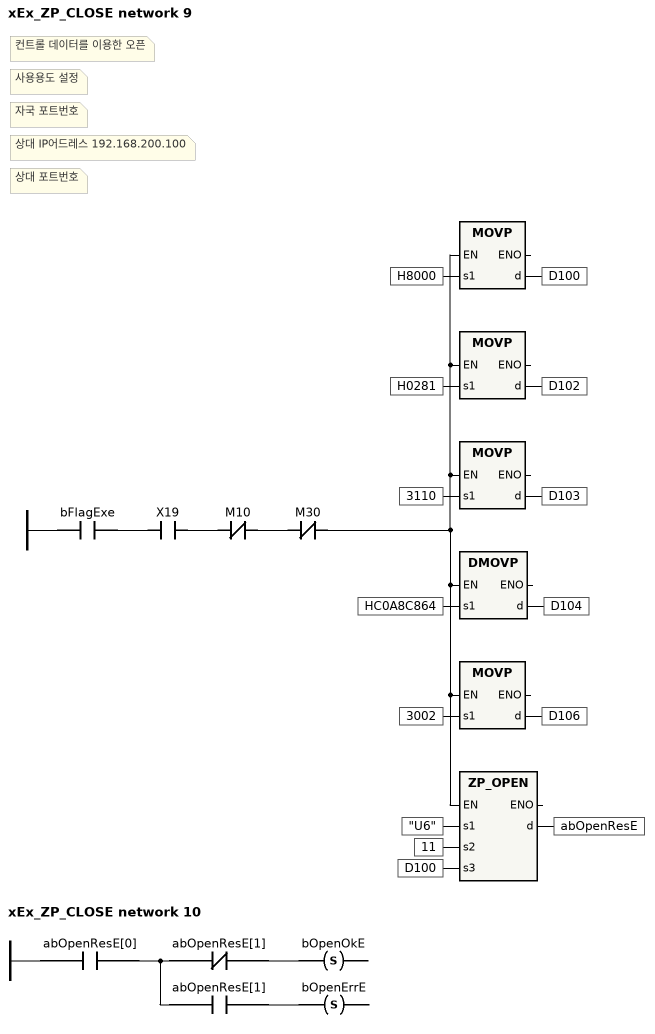
(* network 9 *)
(* 컨트롤 데이터를 이용한 오픈 *)
(* 사용용도 설정 *)
(* 자국 포트번호 *)
(* 상대 IP어드레스 192.168.200.100 *)
(* 상대 포트번호 *)
_p1 := bFlagExe AND X19 AND NOT M10 AND NOT M30;
MOVP(_p1, H8000, D100);
MOVP(_p1, H0281, D102);
MOVP(_p1, 3110, D103);
DMOVP(_p1, HC0A8C864, D104);
MOVP(_p1, 3002, D106);
ZP_OPEN(_p1, "U6", 11, D100, abOpenResE);
(* network 10 *)
SET(abOpenResE[0] AND NOT abOpenResE[1], bOpenOkE);
SET(abOpenResE[0] AND abOpenResE[1], bOpenErrE);
END_PROGRAM

PROGRAM ExEactBUFRCVS
VAR
  bOpenReqC : BOOL;
  bCsetReq : BOOL;
  bOpenReqE : BOOL;
  bOpenOkC : BOOL;
  bOpenOkE : BOOL;
  bOpenErrC : BOOL;
  bOpenErrE : BOOL;
  abOpenResC : ARRAY [0..1] OF BOOL;
  abOpenResE : ARRAY [0..1] OF BOOL;
  acOpenDataC : ARRAY [0..9] OF INT;
  acCsetData : ARRAY [0..4] OF INT;
  acRdCtrl : ARRAY [0..9] OF INT;
  bSendReqC : BOOL;
  bSendReqE : BOOL;
  bSendOkC : BOOL;
  bSendOkE : BOOL;
  bSendErrC : BOOL;
  bSendErrE : BOOL;
  abSendResC : ARRAY [0..1] OF BOOL;
  abSendResE : ARRAY [0..1] OF BOOL;
  abSendResF : ARRAY [0..1] OF BOOL;
  acSendDataC : ARRAY [0..1] OF INT;
  acSendDataE : ARRAY [0..1] OF INT;
  acSendDataF : ARRAY [0..1] OF INT;
  bRecvOkC : BOOL;
  bRecvOkE : BOOL;
  bRecvOkF : BOOL;
  bRecvErrC : BOOL;
  bRecvErrE : BOOL;
  bRecvErrF : BOOL;
  abRecvResC : ARRAY [0..1] OF BOOL;
  abRecvResE : ARRAY [0..1] OF BOOL;
  abRecvResF : ARRAY [0..1] OF BOOL;
  acRecvDataC : ARRAY [0..1] OF INT;
  acRecvDataE : ARRAY [0..1] OF INT;
  acRecvDataF : ARRAY [0..1] OF INT;
  bCloseReqC : BOOL;
  bCloseOkC : BOOL;
  bCloseOkE : BOOL;
  bCloseErrC : BOOL;
  bCloseErrE : BOOL;
  abCloseResC : ARRAY [0..1] OF BOOL;
  abCloseResE : ARRAY [0..1] OF BOOL;
  acCloseDataC : ARRAY [0..1] OF INT;
  CntSend1 : INT;
  CntSend2 : INT;
  CntSend3 : INT;
  CntRecv1 : INT;
  CntRecvErr1 : INT;
  CntRecv2 : INT;
  CntRecv3 : INT;
  CntRecvErr2 : INT;
  CntRecvErr3 : INT;
  ErrCodeCC : INT;
  ErrCodeSE : INT;
  ErrCodeSF : INT;
  ErrCodeRC : INT;
  ErrCodeRE : INT;
  ErrCodeRF : INT;
  Mov4INT_1 : Mov4INT;
  Mov8INT_1 : Mov8INT;
  Mov4INT_2 : Mov4INT;
  Mov4INT_3 : Mov4INT;
  Mov4INT_4 : Mov4INT;
  Word2Bit8_1 : Word2Bit8;
  Word2Bit8_2 : Word2Bit8;
  Word2Bit8_3 : Word2Bit8;
  Word2Bit8_4 : Word2Bit8;
  Word2Bit8_5 : Word2Bit8;
  Word2Bit8_6 : Word2Bit8;
  TON_1 : TON;
  TON_2 : TON;
  TON_3 : TON;
  Status1 : WORD;
  Status2 : WORD;
  Status3 : WORD;
  Word2Bit16_1 : Word2Bit16;
  Word2Bit16_2 : Word2Bit16;
  Word2Bit16_3 : Word2Bit16;
  acOpenDataE : ARRAY [0..9] OF INT;
  acCloseDataE : ARRAY [0..1] OF INT;
  ErrCodeOE : INT;
  ErrCodeSC : INT;
  ErrCodeCE : INT;
  ErrCodeOC : INT;
  bCloseReqE : BOOL;
  Mov4INT_5 : Mov4INT;
  Mov4INT_6 : Mov4INT;
  Mov4INT_7 : Mov4INT;
  Mov4INT_8 : Mov4INT;
END_VAR
(* structured ladder/FBD written out as ST: instructions are called as NAME(EN, inputs, outputs); _pN, _eN, _tN stand for wires *)
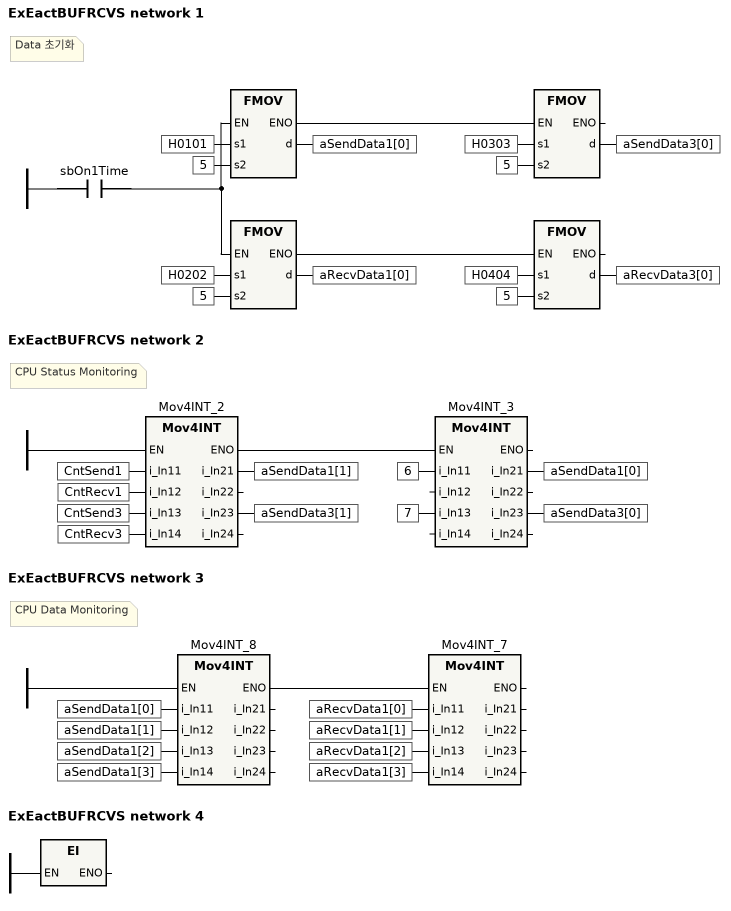
(* network 1 *)
(* Data 초기화 *)
_e1 := FMOV(sbOn1Time, H0101, 5, aSendData1[0]);
FMOV(_e1, H0303, 5, aSendData3[0]);
_e2 := FMOV(sbOn1Time, H0202, 5, aRecvData1[0]);
FMOV(_e2, H0404, 5, aRecvData3[0]);
(* network 2 *)
(* CPU Status Monitoring *)
Mov4INT_2(EN := TRUE, i_In11 := CntSend1, i_In12 := CntRecv1, i_In13 := CntSend3, i_In14 := CntRecv3, i_In21 => aSendData1[1], i_In23 => aSendData3[1]);
Mov4INT_3(EN := Mov4INT_2.ENO, i_In11 := 6, i_In13 := 7, i_In21 => aSendData1[0], i_In23 => aSendData3[0]);
(* network 3 *)
(* CPU Data Monitoring *)
Mov4INT_8(EN := TRUE, i_In11 := aSendData1[0], i_In12 := aSendData1[1], i_In13 := aSendData1[2], i_In14 := aSendData1[3]);
Mov4INT_7(EN := Mov4INT_8.ENO, i_In11 := aRecvData1[0], i_In12 := aRecvData1[1], i_In13 := aRecvData1[2], i_In14 := aRecvData1[3]);
(* network 4 *)
EI(TRUE);
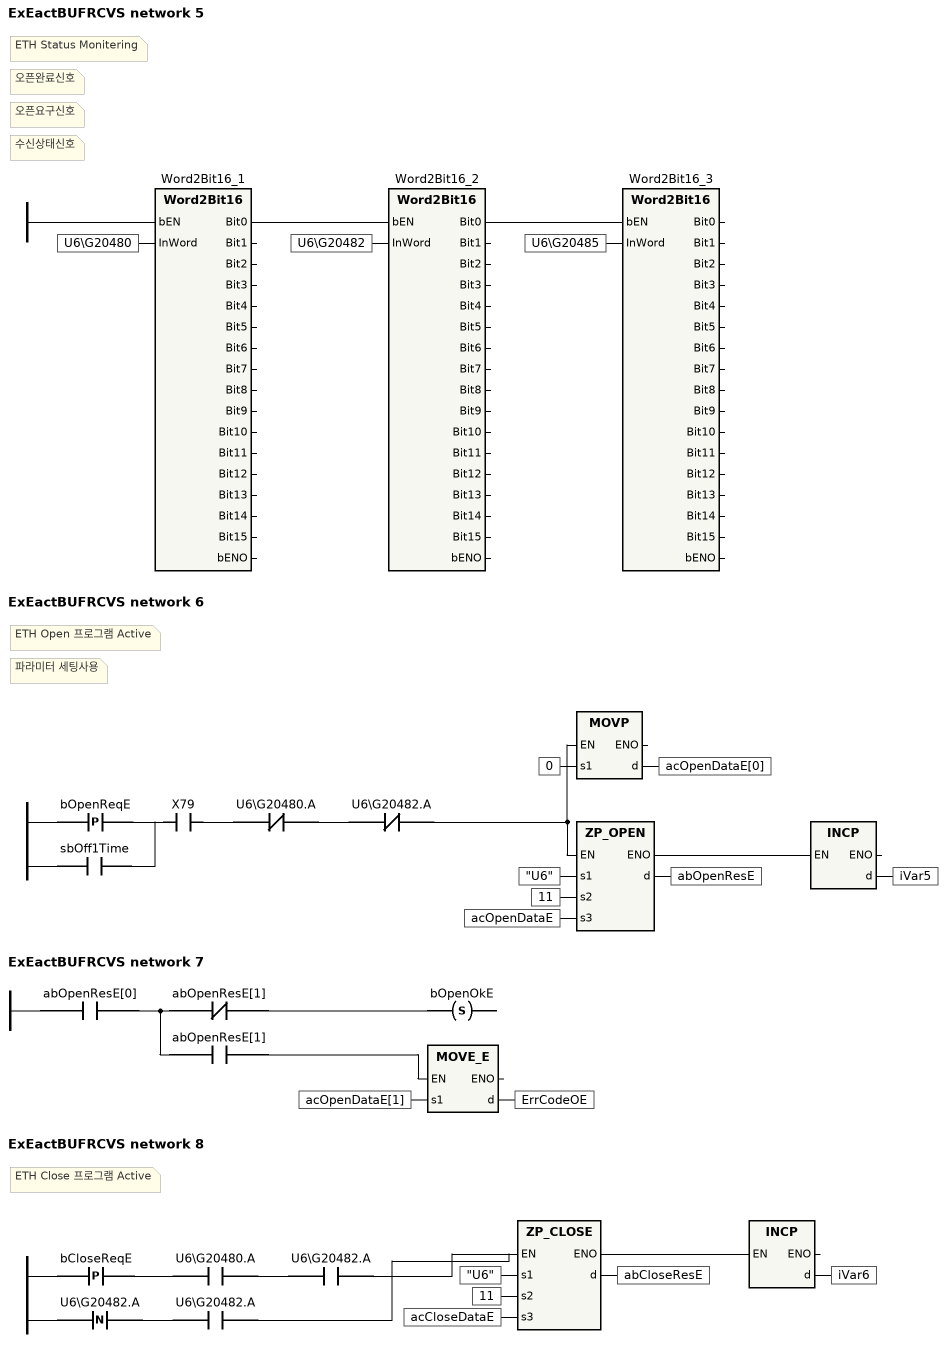
(* network 5 *)
(* ETH Status Monitering *)
(* 오픈완료신호 *)
(* 오픈요구신호 *)
(* 수신상태신호 *)
Word2Bit16_1(bEN := TRUE, InWord := U6\G20480);
Word2Bit16_2(bEN := Word2Bit16_1.Bit0, InWord := U6\G20482);
Word2Bit16_3(bEN := Word2Bit16_2.Bit0, InWord := U6\G20485);
(* network 6 *)
(* ETH Open 프로그램 Active *)
(* 파라미터 세팅사용 *)
_p1 := (((LDP(TRUE, bOpenReqE) OR sbOff1Time) AND X79) AND NOT U6\G20480.A) AND NOT U6\G20482.A;
MOVP(_p1, 0, acOpenDataE[0]);
_e2 := ZP_OPEN(_p1, "U6", 11, acOpenDataE, abOpenResE);
INCP(_e2, iVar5);
(* network 7 *)
SET(abOpenResE[0] AND NOT abOpenResE[1], bOpenOkE);
MOVE_E(abOpenResE[0] AND abOpenResE[1], acOpenDataE[1], ErrCodeOE);
(* network 8 *)
(* ETH Close 프로그램 Active *)
_e1 := ZP_CLOSE((LDP(TRUE, bCloseReqE) AND U6\G20480.A AND U6\G20482.A) OR (LDF(TRUE, U6\G20482.A) AND U6\G20482.A), "U6", 11, acCloseDataE, abCloseResE);
INCP(_e1, iVar6);
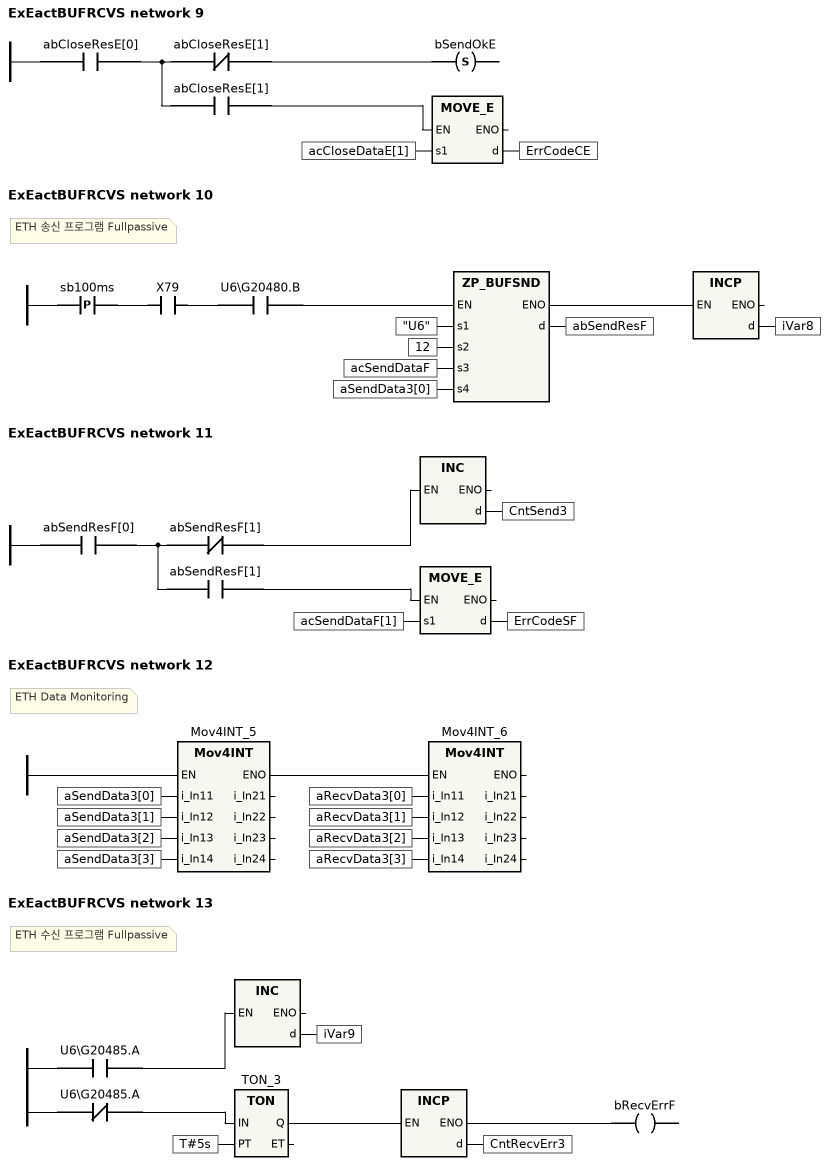
(* network 9 *)
SET(abCloseResE[0] AND NOT abCloseResE[1], bSendOkE);
MOVE_E(abCloseResE[0] AND abCloseResE[1], acCloseDataE[1], ErrCodeCE);
(* network 10 *)
(* ETH 송신 프로그램 Fullpassive *)
_e1 := ZP_BUFSND(LDP(TRUE, sb100ms) AND X79 AND U6\G20480.B, "U6", 12, acSendDataF, aSendData3[0], abSendResF);
INCP(_e1, iVar8);
(* network 11 *)
INC(abSendResF[0] AND NOT abSendResF[1], CntSend3);
MOVE_E(abSendResF[0] AND abSendResF[1], acSendDataF[1], ErrCodeSF);
(* network 12 *)
(* ETH Data Monitoring *)
Mov4INT_5(EN := TRUE, i_In11 := aSendData3[0], i_In12 := aSendData3[1], i_In13 := aSendData3[2], i_In14 := aSendData3[3]);
Mov4INT_6(EN := Mov4INT_5.ENO, i_In11 := aRecvData3[0], i_In12 := aRecvData3[1], i_In13 := aRecvData3[2], i_In14 := aRecvData3[3]);
(* network 13 *)
(* ETH 수신 프로그램 Fullpassive *)
INC(U6\G20485.A, iVar9);
TON_3(IN := NOT U6\G20485.A, PT := T#5s);
_e1 := INCP(TON_3.Q, CntRecvErr3);
bRecvErrF := _e1;
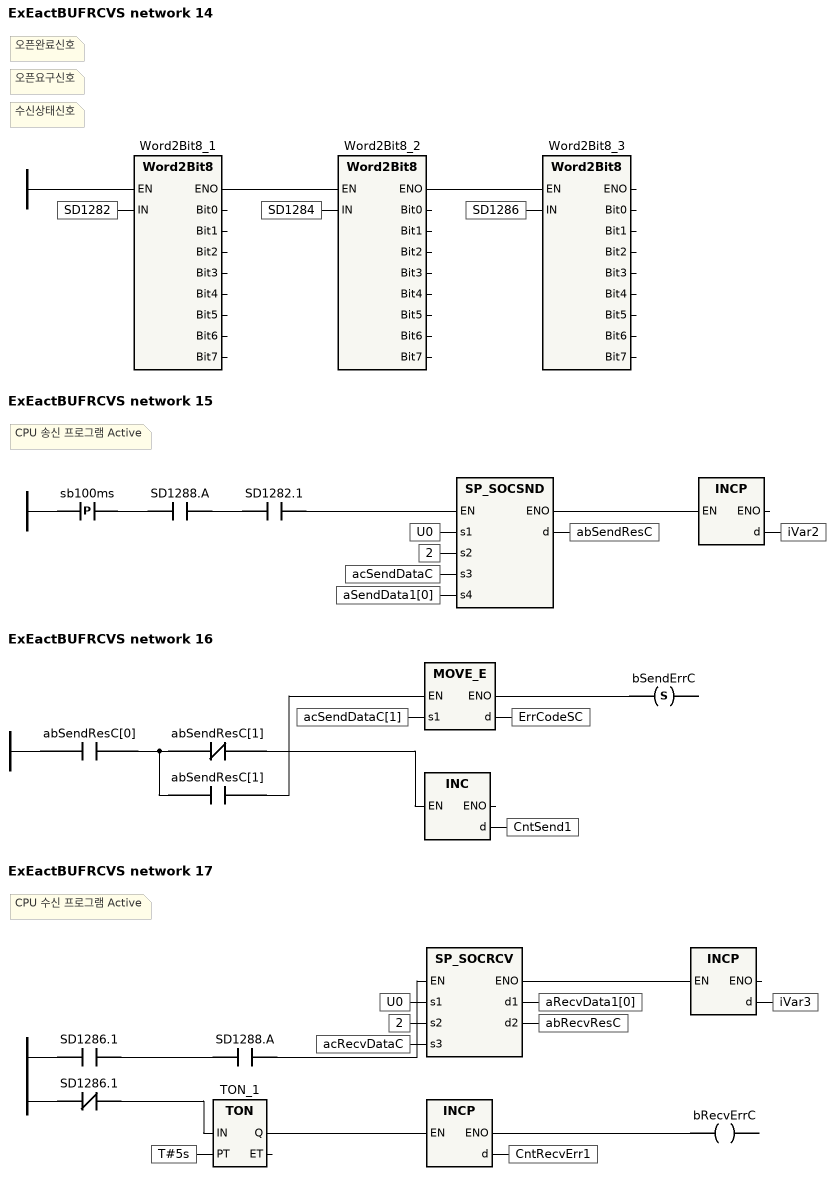
(* network 14 *)
(* 오픈완료신호 *)
(* 오픈요구신호 *)
(* 수신상태신호 *)
Word2Bit8_1(EN := TRUE, IN := SD1282);
Word2Bit8_2(EN := Word2Bit8_1.ENO, IN := SD1284);
Word2Bit8_3(EN := Word2Bit8_2.ENO, IN := SD1286);
(* network 15 *)
(* CPU 송신 프로그램 Active *)
_e1 := SP_SOCSND(LDP(TRUE, sb100ms) AND SD1288.A AND SD1282.1, U0, 2, acSendDataC, aSendData1[0], abSendResC);
INCP(_e1, iVar2);
(* network 16 *)
INC(abSendResC[0] AND NOT abSendResC[1], CntSend1);
_e1 := MOVE_E(abSendResC[0] AND abSendResC[1], acSendDataC[1], ErrCodeSC);
SET(_e1, bSendErrC);
(* network 17 *)
(* CPU 수신 프로그램 Active *)
_e1 := SP_SOCRCV(SD1286.1 AND SD1288.A, U0, 2, acRecvDataC, aRecvData1[0], abRecvResC);
INCP(_e1, iVar3);
TON_1(IN := NOT SD1286.1, PT := T#5s);
_e2 := INCP(TON_1.Q, CntRecvErr1);
bRecvErrC := _e2;
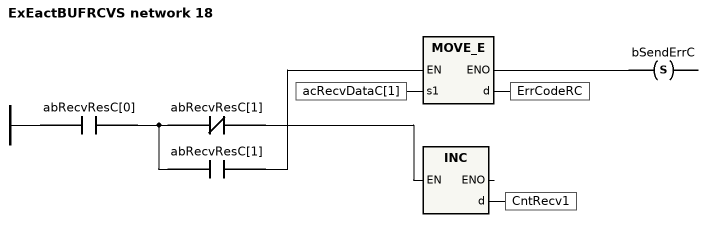
(* network 18 *)
INC(abRecvResC[0] AND NOT abRecvResC[1], CntRecv1);
_e1 := MOVE_E(abRecvResC[0] AND abRecvResC[1], acRecvDataC[1], ErrCodeRC);
SET(_e1, bSendErrC);
END_PROGRAM

PROGRAM ExEact_INT
VAR
  bOpenReqC : BOOL;
  bCsetReq : BOOL;
  bOpenReqE : BOOL;
  bOpenOkC : BOOL;
  bOpenOkE : BOOL;
  bOpenErrC : BOOL;
  bOpenErrE : BOOL;
  abOpenResC : ARRAY [0..1] OF BOOL;
  abOpenResE : ARRAY [0..1] OF BOOL;
  acOpenDataC : ARRAY [0..9] OF INT;
  acCsetData : ARRAY [0..4] OF INT;
  acRdCtrl : ARRAY [0..9] OF INT;
  bSendReqC : BOOL;
  bSendReqE : BOOL;
  bSendOkC : BOOL;
  bSendOkE : BOOL;
  bSendErrC : BOOL;
  bSendErrE : BOOL;
  abSendResC : ARRAY [0..1] OF BOOL;
  abSendResE : ARRAY [0..1] OF BOOL;
  abSendResF : ARRAY [0..1] OF BOOL;
  acSendDataC : ARRAY [0..1] OF INT;
  acSendDataE : ARRAY [0..1] OF INT;
  acSendDataF : ARRAY [0..1] OF INT;
  bRecvOkC : BOOL;
  bRecvOkE : BOOL;
  bRecvOkF : BOOL;
  bRecvErrC : BOOL;
  bRecvErrE : BOOL;
  bRecvErrF : BOOL;
  abRecvResC : ARRAY [0..1] OF BOOL;
  abRecvResE : ARRAY [0..1] OF BOOL;
  abRecvResF : ARRAY [0..1] OF BOOL;
  acRecvDataC : ARRAY [0..1] OF INT;
  acRecvDataE : ARRAY [0..1] OF INT;
  acRecvDataF : ARRAY [0..1] OF INT;
  bCloseReqC : BOOL;
  bCloseOkC : BOOL;
  bCloseOkE : BOOL;
  bCloseErrC : BOOL;
  bCloseErrE : BOOL;
  abCloseResC : ARRAY [0..1] OF BOOL;
  abCloseResE : ARRAY [0..1] OF BOOL;
  acCloseDataC : ARRAY [0..1] OF INT;
  CntSend1 : INT;
  CntSend2 : INT;
  CntSend3 : INT;
  CntRecv1 : INT;
  CntRecvErr1 : INT;
  CntRecv2 : INT;
  CntRecv3 : INT;
  CntRecvErr2 : INT;
  CntRecvErr3 : INT;
  ErrCodeCC : INT;
  ErrCodeSE : INT;
  ErrCodeSF : INT;
  ErrCodeRC : INT;
  ErrCodeRE : INT;
  ErrCodeRF : INT;
  Mov4INT_1 : Mov4INT;
  Mov8INT_1 : Mov8INT;
  Mov4INT_2 : Mov4INT;
  Mov4INT_3 : Mov4INT;
  Mov4INT_4 : Mov4INT;
  Word2Bit8_1 : Word2Bit8;
  Word2Bit8_2 : Word2Bit8;
  Word2Bit8_3 : Word2Bit8;
  Word2Bit8_4 : Word2Bit8;
  Word2Bit8_5 : Word2Bit8;
  Word2Bit8_6 : Word2Bit8;
  TON_1 : TON;
  TON_2 : TON;
  TON_3 : TON;
  Status1 : WORD;
  Status2 : WORD;
  Status3 : WORD;
  Word2Bit16_1 : Word2Bit16;
  Word2Bit16_2 : Word2Bit16;
  Word2Bit16_3 : Word2Bit16;
  acOpenDataE : ARRAY [0..9] OF INT;
  acCloseDataE : ARRAY [0..1] OF INT;
  ErrCodeOE : INT;
  ErrCodeSC : INT;
  ErrCodeCE : INT;
  ErrCodeOC : INT;
  bCloseReqE : BOOL;
  Mov4INT_5 : Mov4INT;
  Mov4INT_6 : Mov4INT;
  Mov4INT_7 : Mov4INT;
  Mov4INT_8 : Mov4INT;
END_VAR
(* structured ladder/FBD written out as ST: instructions are called as NAME(EN, inputs, outputs); _pN, _eN, _tN stand for wires *)
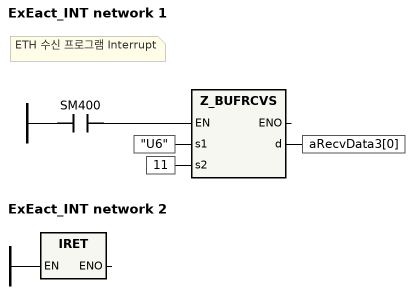
(* network 1 *)
(* ETH 수신 프로그램 Interrupt *)
Z_BUFRCVS(SM400, "U6", 11, aRecvData3[0]);
(* network 2 *)
IRET(TRUE);
END_PROGRAM

PROGRAM ExERRRD
VAR
  bReqFlag : BOOL;
  bFlagExe : BOOL;
  abComp : ARRAY [0..1] OF BOOL;
  aCtrlData : ARRAY [0..7] OF INT;
  iErrCode : INT;
  iErrInfo : INT;
END_VAR
(* structured ladder/FBD written out as ST: instructions are called as NAME(EN, inputs, outputs); _pN, _eN, _tN stand for wires *)
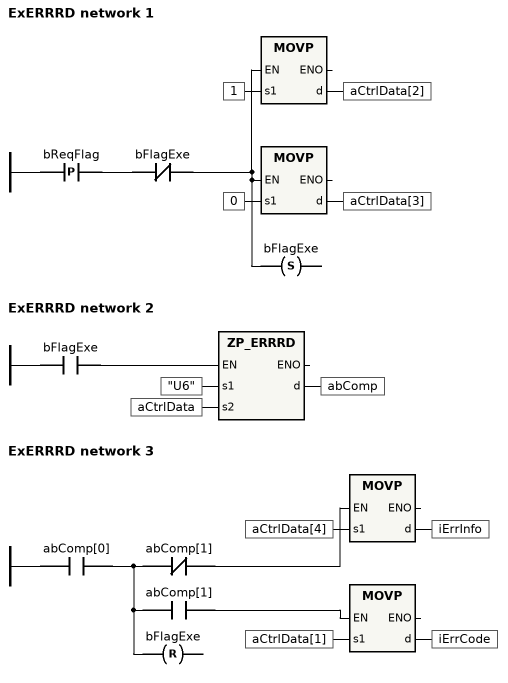
(* network 1 *)
_p1 := LDP(TRUE, bReqFlag) AND NOT bFlagExe;
MOVP(_p1, 1, aCtrlData[2]);
MOVP(_p1, 0, aCtrlData[3]);
SET(_p1, bFlagExe);
(* network 2 *)
ZP_ERRRD(bFlagExe, "U6", aCtrlData, abComp);
(* network 3 *)
MOVP(abComp[0] AND NOT abComp[1], aCtrlData[4], iErrInfo);
MOVP(abComp[0] AND abComp[1], aCtrlData[1], iErrCode);
RST(abComp[0], bFlagExe);
END_PROGRAM

PROGRAM ExUINI2
VAR
  bReqFlag : BOOL;
  bFlagExe : BOOL;
  abComp : ARRAY [0..1] OF BOOL;
  aCtrlData : ARRAY [0..9] OF INT;
  iErrCode : INT;
  bInitExe : BOOL;
  bInitComp : BOOL;
  bInitError : BOOL;
  bInitComp2 : BOOL;
  bInitError2 : BOOL;
  bInitCompEnd : BOOL;
  bCmdInit : BOOL;
  bSetMode : BOOL;
END_VAR
(* structured ladder/FBD written out as ST: instructions are called as NAME(EN, inputs, outputs); _pN, _eN, _tN stand for wires *)
